Yaskawa INFORM job: u_tourne2TRJ3.JBI

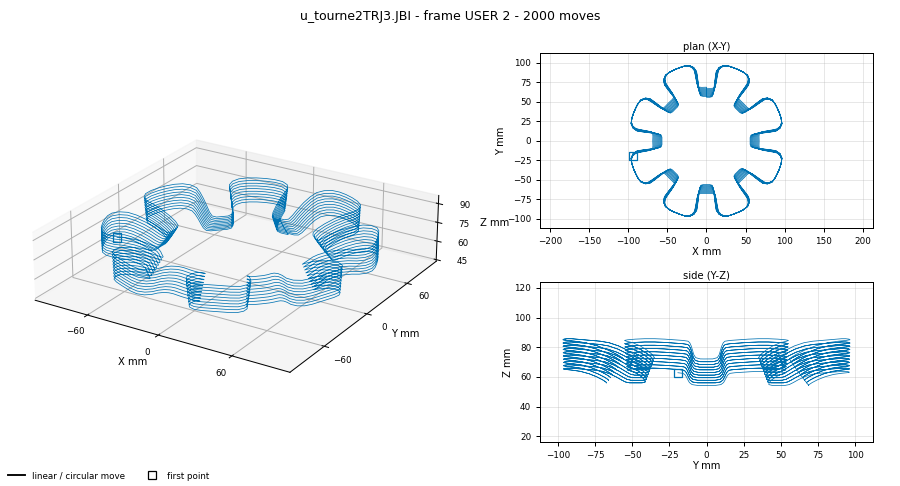
[picture p0: tool path of u_tourne2TRJ3.JBI in frame USER 2, 2000 of 2000 moves have a stored position in this frame; points joined in program order, loops and branches not executed]
/JOB
//NAME u_tourne2TRJ3
///FOLDERNAME DEMO
//POS
///NPOS 2000,0,0,0,0,0
///USER 2
///TOOL 7
///POSTYPE USER
///RECTAN
///RCONF 1,0,0,0,0,0,0,0,0,0,0,0,0,0,0,0,0,0,0,0,0,0,0,0
C00000=-94.423,-19.246,62.877,177.2934,-4.1506,0.0000
C00001=-90.636,-15.942,62.469,172.7027,-3.4329,0.0000
C00002=-85.405,-14.621,61.698,172.2436,-1.7928,0.0000
C00003=-79.780,-13.569,60.151,174.0288,-1.3194,0.0000
C00004=-74.809,-12.586,58.158,176.9959,-0.7631,0.0000
C00005=-71.127,-11.507,56.252,-176.5767,1.2628,0.0000
C00006=-69.044,-9.699,54.888,-163.7827,26.3506,0.0000
C00007=-68.619,-6.200,54.350,-178.9486,38.3072,0.0000
C00008=-68.781,-2.945,54.326,177.7373,38.7538,0.0000
C00009=-68.843,0.000,54.342,180.0000,38.7770,0.0000
C00010=-68.781,2.945,54.326,-177.7373,38.7538,0.0000
C00011=-68.619,6.200,54.350,178.9486,38.3072,0.0000
C00012=-69.044,9.699,54.888,163.7827,26.3559,0.0000
C00013=-71.127,11.507,56.252,176.5767,1.2628,0.0000
C00014=-74.809,12.586,58.158,-176.9959,-0.7631,0.0000
C00015=-79.780,13.569,60.151,-174.0288,-1.3194,0.0000
C00016=-85.405,14.621,61.698,-172.2436,-1.7928,0.0000
C00017=-90.636,15.942,62.469,-172.7027,-3.4329,0.0000
C00018=-94.423,19.246,62.877,-177.2934,-4.1506,0.0000
C00019=-96.154,24.159,63.210,-179.7477,-2.4644,0.0000
C00020=-95.429,29.718,63.547,179.9542,-0.1490,0.0000
C00021=-93.512,35.416,63.770,179.9943,-0.0172,0.0000
C00022=-91.166,41.080,63.770,179.9943,-0.0172,0.0000
C00023=-88.493,46.465,63.547,179.9255,-0.1375,0.0000
C00024=-85.074,50.908,63.210,178.0796,-1.5652,0.0000
C00025=-80.376,53.158,62.877,175.1578,-1.0293,0.0000
C00026=-75.362,52.817,62.469,172.4296,2.7522,0.0000
C00027=-70.729,50.052,61.698,173.2455,4.2443,0.0000
C00028=-66.007,46.818,60.151,174.8393,3.3040,0.0000
C00029=-61.798,43.998,58.158,177.3394,1.5891,0.0000
C00030=-58.431,42.158,56.252,-176.6911,-1.5268,0.0000
C00031=-55.679,41.963,54.888,-150.9263,8.2291,0.0000
C00032=-52.905,44.137,54.350,-150.2465,28.6181,0.0000
C00033=-50.718,46.553,54.326,-151.6440,30.7742,0.0000
C00034=-48.679,48.679,54.342,-150.4041,29.6014,0.0000
C00035=-46.553,50.718,54.326,-149.2258,28.3560,0.0000
C00036=-44.137,52.905,54.350,-151.3819,29.7535,0.0000
C00037=-41.963,55.680,54.888,-171.7709,29.0737,0.0000
C00038=-42.158,58.431,56.252,178.4732,3.3089,0.0000
C00039=-43.998,61.798,58.158,-178.4109,-2.6606,0.0000
C00040=-46.818,66.007,60.151,-176.6960,-5.1607,0.0000
C00041=-50.052,70.729,61.698,-175.7557,-6.7545,0.0000
C00042=-52.817,75.362,62.469,-177.2478,-7.5704,0.0000
C00043=-53.158,80.376,62.877,178.9707,-4.8422,0.0000
C00044=-50.908,85.074,63.210,178.4348,-1.9204,0.0000
C00045=-46.465,88.493,63.547,179.8625,-0.0745,0.0000
C00046=-41.080,91.166,63.770,179.9828,-0.0057,0.0000
C00047=-35.416,93.512,63.770,179.9828,-0.0057,0.0000
C00048=-29.718,95.429,63.547,179.8510,-0.0458,0.0000
C00049=-24.159,96.154,63.210,177.5356,0.2523,0.0000
C00050=-19.246,94.423,62.877,175.8494,2.7066,0.0000
C00051=-15.942,90.636,62.469,176.5671,7.2973,0.0000
C00052=-14.621,85.405,61.698,178.2072,7.7564,0.0000
C00053=-13.569,79.780,60.151,178.6806,5.9712,0.0000
C00054=-12.586,74.809,58.158,179.2369,3.0041,0.0000
C00055=-11.507,71.127,56.252,-178.7372,-3.4233,0.0000
C00056=-9.699,69.044,54.888,-153.6441,-16.2173,0.0000
C00057=-6.200,68.619,54.350,-141.6928,-1.0514,0.0000
C00058=-2.945,68.781,54.326,-141.2462,2.2627,0.0000
C00059=0.000,68.843,54.342,-141.2230,-0.0000,0.0000
C00060=0.000,67.469,56.061,-141.5406,-0.0000,0.0000
C00061=2.820,67.413,56.044,-141.5604,-2.2018,0.0000
C00062=5.989,67.263,56.069,-142.0562,1.4094,0.0000
C00063=9.441,67.734,56.637,-154.9623,16.3637,0.0000
C00064=11.191,69.937,58.076,-179.1454,2.5050,0.0000
C00065=12.227,73.809,60.085,179.1965,-3.3826,0.0000
C00066=13.183,79.025,62.181,178.7265,-6.0864,0.0000
C00067=14.211,84.918,63.804,178.3230,-7.7443,0.0000
C00068=15.500,90.396,64.610,176.7346,-7.3136,0.0000
C00069=18.832,94.373,65.037,175.8895,-2.7812,0.0000
C00070=23.832,96.213,65.385,177.5470,-0.2753,0.0000
C00071=29.513,95.497,65.736,179.8453,0.0458,0.0000
C00072=35.347,93.539,65.969,179.9828,0.0057,0.0000
C00073=41.148,91.136,65.969,179.9828,0.0057,0.0000
C00074=46.658,88.395,65.736,179.8625,0.0745,0.0000
C00075=51.181,84.885,65.385,178.4577,1.9261,0.0000
C00076=53.416,80.048,65.037,179.0569,4.8707,0.0000
C00077=52.959,74.880,64.610,-177.1154,7.4730,0.0000
C00078=49.997,70.095,63.804,-175.6871,6.6682,0.0000
C00079=46.557,65.200,62.181,-176.5862,5.2074,0.0000
C00080=43.545,60.837,60.085,-178.1753,2.9592,0.0000
C00081=41.540,57.367,58.076,178.8300,-2.3790,0.0000
C00082=41.220,54.571,56.637,-173.0071,-28.2766,0.0000
C00083=43.327,51.796,56.069,-151.9011,-29.6258,0.0000
C00084=45.674,49.662,56.044,-149.5306,-28.1040,0.0000
C00085=47.708,47.708,56.061,-150.6808,-29.3192,0.0000
C00086=49.662,45.674,56.044,-151.8960,-30.4694,0.0000
C00087=51.797,43.327,56.069,-150.3742,-28.0989,0.0000
C00088=54.571,41.220,56.637,-151.7234,-6.9929,0.0000
C00089=57.367,41.540,58.076,-177.6210,1.1700,0.0000
C00090=60.837,43.545,60.085,177.0408,-1.8247,0.0000
C00091=65.200,46.557,62.181,174.7926,-3.4138,0.0000
C00092=70.095,49.997,63.804,173.3318,-4.3129,0.0000
C00093=74.880,52.959,64.610,172.5270,-2.8846,0.0000
C00094=80.048,53.416,65.037,175.1293,0.9431,0.0000
C00095=84.885,51.181,65.385,178.0739,1.5423,0.0000
C00096=88.395,46.658,65.736,179.9255,0.1375,0.0000
C00097=91.136,41.148,65.969,179.9943,0.0172,0.0000
C00098=93.539,35.347,65.969,179.9943,0.0172,0.0000
C00099=95.497,29.513,65.736,179.9542,0.1547,0.0000
C00100=96.213,23.832,65.385,-179.7247,2.4530,0.0000
C00101=94.373,18.832,65.037,-177.2188,4.1105,0.0000
C00102=90.396,15.500,64.610,-172.6864,3.2654,0.0000
C00103=84.918,14.211,63.804,-172.2557,1.6770,0.0000
C00104=79.025,13.183,62.181,-173.9136,1.2735,0.0000
C00105=73.809,12.227,60.085,-176.6174,0.8035,0.0000
C00106=69.937,11.191,58.076,177.4950,-0.8546,0.0000
C00107=67.734,9.441,56.637,163.6363,-25.0377,0.0000
C00108=67.263,5.989,56.069,178.5906,-37.9438,0.0000
C00109=67.413,2.820,56.044,-177.7982,-38.4396,0.0000
C00110=67.469,0.000,56.061,-180.0000,-38.4594,0.0000
C00111=67.413,-2.820,56.044,177.7982,-38.4396,0.0000
C00112=67.263,-5.989,56.069,-178.5906,-37.9438,0.0000
C00113=67.734,-9.441,56.637,-163.6363,-25.0377,0.0000
C00114=69.937,-11.191,58.076,-177.4950,-0.8546,0.0000
C00115=73.809,-12.227,60.085,176.6174,0.8035,0.0000
C00116=79.025,-13.183,62.181,173.9136,1.2735,0.0000
C00117=84.918,-14.211,63.804,172.2557,1.6770,0.0000
C00118=90.396,-15.500,64.610,172.6864,3.2654,0.0000
C00119=94.373,-18.832,65.037,177.2188,4.1105,0.0000
C00120=96.213,-23.832,65.385,179.7247,2.4530,0.0000
C00121=95.497,-29.513,65.736,-179.9542,0.1547,0.0000
C00122=93.539,-35.347,65.969,-179.9943,0.0172,0.0000
C00123=91.136,-41.148,65.969,-179.9943,0.0172,0.0000
C00124=88.395,-46.658,65.736,-179.9255,0.1375,0.0000
C00125=84.885,-51.181,65.385,-178.0739,1.5423,0.0000
C00126=80.048,-53.416,65.037,-175.1293,0.9431,0.0000
C00127=74.880,-52.959,64.610,-172.5270,-2.8846,0.0000
C00128=70.095,-49.997,63.804,-173.3318,-4.3129,0.0000
C00129=65.200,-46.557,62.181,-174.7926,-3.4138,0.0000
C00130=60.837,-43.545,60.085,-177.0408,-1.8247,0.0000
C00131=57.367,-41.540,58.076,177.6210,1.1700,0.0000
C00132=54.571,-41.220,56.637,151.7234,-6.9929,0.0000
C00133=51.796,-43.327,56.069,150.3742,-28.0989,0.0000
C00134=49.662,-45.674,56.044,151.8960,-30.4694,0.0000
C00135=47.708,-47.708,56.061,150.6808,-29.3192,0.0000
C00136=45.674,-49.662,56.044,149.5306,-28.1040,0.0000
C00137=43.327,-51.797,56.069,151.9011,-29.6258,0.0000
C00138=41.220,-54.571,56.637,173.0071,-28.2766,0.0000
C00139=41.540,-57.367,58.076,-178.8300,-2.3790,0.0000
C00140=43.545,-60.837,60.085,178.1753,2.9592,0.0000
C00141=46.557,-65.200,62.181,176.5862,5.2074,0.0000
C00142=49.997,-70.095,63.804,175.6871,6.6682,0.0000
C00143=52.959,-74.880,64.610,177.1154,7.4730,0.0000
C00144=53.416,-80.048,65.037,-179.0569,4.8707,0.0000
C00145=51.181,-84.885,65.385,-178.4577,1.9261,0.0000
C00146=46.658,-88.395,65.736,-179.8625,0.0745,0.0000
C00147=41.148,-91.136,65.969,-179.9828,0.0057,0.0000
C00148=35.347,-93.539,65.969,-179.9828,0.0057,0.0000
C00149=29.513,-95.497,65.736,-179.8453,0.0458,0.0000
C00150=23.832,-96.213,65.385,-177.5470,-0.2753,0.0000
C00151=18.832,-94.373,65.037,-175.8895,-2.7812,0.0000
C00152=15.500,-90.396,64.610,-176.7346,-7.3136,0.0000
C00153=14.211,-84.918,63.804,-178.3230,-7.7443,0.0000
C00154=13.183,-79.025,62.181,-178.7265,-6.0864,0.0000
C00155=12.227,-73.809,60.085,-179.1965,-3.3826,0.0000
C00156=11.191,-69.937,58.076,179.1454,2.5050,0.0000
C00157=9.441,-67.734,56.637,154.9623,16.3637,0.0000
C00158=5.989,-67.263,56.069,142.0562,1.4094,0.0000
C00159=2.820,-67.413,56.044,141.5604,-2.2018,0.0000
C00160=0.000,-67.469,56.061,141.5406,-0.0000,0.0000
C00161=0.000,-67.469,56.061,141.5406,-0.0000,0.0000
C00162=-2.820,-67.413,56.044,141.5604,2.2018,0.0000
C00163=-5.989,-67.263,56.069,142.0562,-1.4094,0.0000
C00164=-9.441,-67.734,56.637,154.9623,-16.3637,0.0000
C00165=-11.191,-69.937,58.076,179.1454,-2.5050,0.0000
C00166=-12.227,-73.809,60.085,-179.1965,3.3826,0.0000
C00167=-13.183,-79.025,62.181,-178.7265,6.0864,0.0000
C00168=-14.211,-84.918,63.804,-178.3230,7.7443,0.0000
C00169=-15.500,-90.396,64.610,-176.7346,7.3136,0.0000
C00170=-18.832,-94.373,65.037,-175.8895,2.7812,0.0000
C00171=-23.832,-96.213,65.385,-177.5470,0.2753,0.0000
C00172=-29.513,-95.497,65.736,-179.8453,-0.0458,0.0000
C00173=-35.347,-93.539,65.969,-179.9828,-0.0057,0.0000
C00174=-41.148,-91.136,65.969,-179.9828,-0.0057,0.0000
C00175=-46.658,-88.395,65.736,-179.8625,-0.0745,0.0000
C00176=-51.181,-84.885,65.385,-178.4577,-1.9261,0.0000
C00177=-53.416,-80.048,65.037,-179.0569,-4.8707,0.0000
C00178=-52.959,-74.880,64.610,177.1154,-7.4730,0.0000
C00179=-49.997,-70.095,63.804,175.6871,-6.6682,0.0000
C00180=-46.557,-65.200,62.181,176.5862,-5.2074,0.0000
C00181=-43.545,-60.837,60.085,178.1753,-2.9592,0.0000
C00182=-41.540,-57.367,58.076,-178.8300,2.3790,0.0000
C00183=-41.220,-54.571,56.637,173.0071,28.2766,0.0000
C00184=-43.327,-51.796,56.069,151.9011,29.6258,0.0000
C00185=-45.674,-49.662,56.044,149.5306,28.1040,0.0000
C00186=-47.708,-47.708,56.061,150.6808,29.3192,0.0000
C00187=-49.662,-45.674,56.044,151.8960,30.4694,0.0000
C00188=-51.797,-43.327,56.069,150.3742,28.0989,0.0000
C00189=-54.571,-41.220,56.637,151.7234,6.9929,0.0000
C00190=-57.367,-41.540,58.076,177.6210,-1.1700,0.0000
C00191=-60.837,-43.545,60.085,-177.0408,1.8247,0.0000
C00192=-65.200,-46.557,62.181,-174.7926,3.4138,0.0000
C00193=-70.095,-49.997,63.804,-173.3318,4.3129,0.0000
C00194=-74.880,-52.959,64.610,-172.5270,2.8846,0.0000
C00195=-80.048,-53.416,65.037,-175.1293,-0.9431,0.0000
C00196=-84.885,-51.181,65.385,-178.0739,-1.5423,0.0000
C00197=-88.395,-46.658,65.736,-179.9255,-0.1375,0.0000
C00198=-91.136,-41.148,65.969,-179.9943,-0.0172,0.0000
C00199=-93.539,-35.347,65.969,-179.9943,-0.0172,0.0000
C00200=-95.497,-29.513,65.736,-179.9542,-0.1547,0.0000
C00201=-96.213,-23.832,65.385,179.7247,-2.4530,0.0000
C00202=-94.373,-18.832,65.037,177.2188,-4.1105,0.0000
C00203=-90.396,-15.500,64.610,172.6864,-3.2654,0.0000
C00204=-84.918,-14.211,63.804,172.2557,-1.6770,0.0000
C00205=-79.025,-13.183,62.181,173.9136,-1.2735,0.0000
C00206=-73.809,-12.227,60.085,176.6174,-0.8035,0.0000
C00207=-69.937,-11.191,58.076,-177.4950,0.8546,0.0000
C00208=-67.734,-9.441,56.637,-163.6363,25.0377,0.0000
C00209=-67.263,-5.989,56.069,-178.5906,37.9438,0.0000
C00210=-67.413,-2.820,56.044,177.7982,38.4396,0.0000
C00211=-67.469,0.000,56.061,180.0000,38.4594,0.0000
C00212=-67.413,2.820,56.044,-177.7982,38.4396,0.0000
C00213=-67.263,5.989,56.069,178.5906,37.9438,0.0000
C00214=-67.734,9.441,56.637,163.6363,25.0377,0.0000
C00215=-69.937,11.191,58.076,177.4950,0.8546,0.0000
C00216=-73.809,12.227,60.085,-176.6174,-0.8035,0.0000
C00217=-79.025,13.183,62.181,-173.9136,-1.2735,0.0000
C00218=-84.918,14.211,63.804,-172.2557,-1.6770,0.0000
C00219=-90.396,15.500,64.610,-172.6864,-3.2654,0.0000
C00220=-94.373,18.832,65.037,-177.2188,-4.1105,0.0000
C00221=-96.213,23.832,65.385,-179.7247,-2.4530,0.0000
C00222=-95.497,29.513,65.736,179.9542,-0.1547,0.0000
C00223=-93.539,35.347,65.969,179.9943,-0.0172,0.0000
C00224=-91.136,41.148,65.969,179.9943,-0.0172,0.0000
C00225=-88.395,46.658,65.736,179.9255,-0.1375,0.0000
C00226=-84.885,51.181,65.385,178.0739,-1.5423,0.0000
C00227=-80.048,53.416,65.037,175.1293,-0.9431,0.0000
C00228=-74.880,52.959,64.610,172.5270,2.8846,0.0000
C00229=-70.095,49.997,63.804,173.3318,4.3129,0.0000
C00230=-65.200,46.557,62.181,174.7926,3.4138,0.0000
C00231=-60.837,43.545,60.085,177.0408,1.8247,0.0000
C00232=-57.367,41.540,58.076,-177.6210,-1.1700,0.0000
C00233=-54.571,41.220,56.637,-151.7234,6.9929,0.0000
C00234=-51.796,43.327,56.069,-150.3742,28.0989,0.0000
C00235=-49.662,45.674,56.044,-151.8960,30.4694,0.0000
C00236=-47.708,47.708,56.061,-150.6808,29.3192,0.0000
C00237=-45.674,49.662,56.044,-149.5306,28.1040,0.0000
C00238=-43.327,51.797,56.069,-151.9011,29.6258,0.0000
C00239=-41.220,54.571,56.637,-173.0071,28.2766,0.0000
C00240=-41.540,57.367,58.076,178.8300,2.3790,0.0000
C00241=-43.545,60.837,60.085,-178.1753,-2.9592,0.0000
C00242=-46.557,65.200,62.181,-176.5862,-5.2074,0.0000
C00243=-49.997,70.095,63.804,-175.6871,-6.6682,0.0000
C00244=-52.959,74.880,64.610,-177.1154,-7.4730,0.0000
C00245=-53.416,80.048,65.037,179.0569,-4.8707,0.0000
C00246=-51.181,84.885,65.385,178.4577,-1.9261,0.0000
C00247=-46.658,88.395,65.736,179.8625,-0.0745,0.0000
C00248=-41.148,91.136,65.969,179.9828,-0.0057,0.0000
C00249=-35.347,93.539,65.969,179.9828,-0.0057,0.0000
C00250=-29.513,95.497,65.736,179.8453,-0.0458,0.0000
C00251=-23.832,96.213,65.385,177.5470,0.2753,0.0000
C00252=-18.832,94.373,65.037,175.8895,2.7812,0.0000
C00253=-15.500,90.396,64.610,176.7346,7.3136,0.0000
C00254=-14.211,84.918,63.804,178.3230,7.7443,0.0000
C00255=-13.183,79.025,62.181,178.7265,6.0864,0.0000
C00256=-12.227,73.809,60.085,179.1965,3.3826,0.0000
C00257=-11.191,69.937,58.076,-179.1454,-2.5050,0.0000
C00258=-9.441,67.734,56.637,-154.9623,-16.3637,0.0000
C00259=-5.989,67.263,56.069,-142.0562,-1.4094,0.0000
C00260=-2.820,67.413,56.044,-141.5604,2.2018,0.0000
C00261=0.000,67.469,56.061,-141.5406,-0.0000,0.0000
C00262=0.000,66.107,57.788,-141.9406,-0.0000,0.0000
C00263=2.695,66.055,57.771,-141.9641,-2.1313,0.0000
C00264=5.779,65.917,57.797,-142.5065,1.7619,0.0000
C00265=9.185,66.436,58.394,-156.3339,16.3885,0.0000
C00266=10.880,68.762,59.909,-179.4726,1.6677,0.0000
C00267=11.874,72.826,62.021,179.1732,-3.6871,0.0000
C00268=12.805,78.288,64.219,178.7783,-6.1320,0.0000
C00269=13.814,84.445,65.915,178.4331,-7.6575,0.0000
C00270=15.073,90.163,66.756,176.9144,-7.2602,0.0000
C00271=18.432,94.325,67.200,175.9696,-2.8214,0.0000
C00272=23.517,96.271,67.561,177.5814,-0.2925,0.0000
C00273=29.315,95.562,67.927,179.8510,0.0458,0.0000
C00274=35.280,93.564,68.167,179.9828,0.0057,0.0000
C00275=41.213,91.107,68.167,179.9828,0.0057,0.0000
C00276=46.844,88.301,67.927,179.8625,0.0745,0.0000
C00277=51.445,84.703,67.561,178.4978,1.9147,0.0000
C00278=53.664,79.731,67.200,179.1432,4.8422,0.0000
C00279=53.097,74.413,66.756,-177.0297,7.3058,0.0000
C00280=49.944,69.479,65.915,-175.6707,6.5299,0.0000
C00281=46.303,64.413,64.219,-176.5116,5.2017,0.0000
C00282=43.100,59.892,62.021,-177.9738,3.1951,0.0000
C00283=40.929,56.315,59.909,179.1918,-1.5531,0.0000
C00284=40.483,53.472,58.394,-174.1765,-27.3781,0.0000
C00285=42.524,50.697,57.797,-152.4951,-29.4304,0.0000
C00286=44.802,48.614,57.771,-149.9099,-27.7831,0.0000
C00287=46.745,46.745,57.788,-151.0313,-28.9687,0.0000
C00288=48.613,44.802,57.771,-152.2169,-30.0901,0.0000
C00289=50.697,42.524,57.797,-150.5696,-27.4992,0.0000
C00290=53.472,40.483,58.395,-152.6219,-5.8235,0.0000
C00291=56.315,40.929,59.909,-178.4469,0.8082,0.0000
C00292=59.892,43.100,62.021,176.8049,-2.0262,0.0000
C00293=64.413,46.303,64.219,174.7983,-3.4884,0.0000
C00294=69.479,49.944,65.915,173.4701,-4.3293,0.0000
C00295=74.413,53.097,66.756,172.6942,-2.9703,0.0000
C00296=79.731,53.664,67.200,175.1578,0.8568,0.0000
C00297=84.703,51.445,67.561,178.0853,1.5022,0.0000
C00298=88.301,46.844,67.927,179.9255,0.1375,0.0000
C00299=91.107,41.213,68.167,179.9943,0.0172,0.0000
C00300=93.564,35.280,68.167,179.9943,0.0172,0.0000
C00301=95.562,29.315,67.927,179.9542,0.1490,0.0000
C00302=96.271,23.517,67.561,-179.7075,2.4186,0.0000
C00303=94.325,18.432,67.200,-177.1786,4.0304,0.0000
C00304=90.163,15.073,66.756,-172.7398,3.0856,0.0000
C00305=84.445,13.814,65.915,-172.3425,1.5669,0.0000
C00306=78.288,12.805,64.219,-173.8680,1.2217,0.0000
C00307=72.826,11.874,62.021,-176.3129,0.8268,0.0000
C00308=68.762,10.880,59.909,178.3323,-0.5274,0.0000
C00309=66.436,9.185,58.394,163.6115,-23.6661,0.0000
C00310=65.917,5.779,57.797,178.2381,-37.4935,0.0000
C00311=66.055,2.695,57.771,-177.8687,-38.0359,0.0000
C00312=66.107,0.000,57.788,-180.0000,-38.0594,0.0000
C00313=66.055,-2.695,57.771,177.8687,-38.0359,0.0000
C00314=65.917,-5.780,57.797,-178.2308,-37.4935,0.0000
C00315=66.436,-9.185,58.395,-163.6115,-23.6661,0.0000
C00316=68.762,-10.880,59.909,-178.3323,-0.5274,0.0000
C00317=72.826,-11.874,62.021,176.3129,0.8268,0.0000
C00318=78.288,-12.805,64.219,173.8680,1.2217,0.0000
C00319=84.445,-13.814,65.915,172.3425,1.5669,0.0000
C00320=90.163,-15.073,66.756,172.7398,3.0856,0.0000
C00321=94.325,-18.432,67.200,177.1786,4.0304,0.0000
C00322=96.271,-23.517,67.561,179.7075,2.4186,0.0000
C00323=95.562,-29.315,67.927,-179.9542,0.1490,0.0000
C00324=93.564,-35.280,68.167,-179.9943,0.0172,0.0000
C00325=91.107,-41.213,68.167,-179.9943,0.0172,0.0000
C00326=88.301,-46.844,67.927,-179.9255,0.1375,0.0000
C00327=84.703,-51.445,67.561,-178.0853,1.5022,0.0000
C00328=79.731,-53.664,67.200,-175.1578,0.8568,0.0000
C00329=74.413,-53.097,66.756,-172.6942,-2.9703,0.0000
C00330=69.479,-49.944,65.915,-173.4701,-4.3293,0.0000
C00331=64.413,-46.303,64.219,-174.7983,-3.4884,0.0000
C00332=59.892,-43.100,62.021,-176.8049,-2.0262,0.0000
C00333=56.315,-40.929,59.909,178.4469,0.8082,0.0000
C00334=53.472,-40.483,58.394,152.6219,-5.8235,0.0000
C00335=50.697,-42.524,57.797,150.5696,-27.5049,0.0000
C00336=48.614,-44.802,57.771,152.2169,-30.0901,0.0000
C00337=46.745,-46.745,57.788,151.0313,-28.9687,0.0000
C00338=44.802,-48.613,57.771,149.9099,-27.7831,0.0000
C00339=42.524,-50.697,57.797,152.5008,-29.4304,0.0000
C00340=40.483,-53.472,58.395,174.1765,-27.3781,0.0000
C00341=40.929,-56.315,59.909,-179.1918,-1.5531,0.0000
C00342=43.100,-59.892,62.021,177.9738,3.1951,0.0000
C00343=46.303,-64.413,64.219,176.5116,5.2017,0.0000
C00344=49.944,-69.479,65.915,175.6707,6.5299,0.0000
C00345=53.097,-74.413,66.756,177.0297,7.3058,0.0000
C00346=53.664,-79.731,67.200,-179.1432,4.8422,0.0000
C00347=51.445,-84.703,67.561,-178.4978,1.9147,0.0000
C00348=46.844,-88.301,67.927,-179.8625,0.0745,0.0000
C00349=41.213,-91.107,68.167,-179.9828,0.0057,0.0000
C00350=35.280,-93.564,68.167,-179.9828,0.0057,0.0000
C00351=29.315,-95.562,67.927,-179.8510,0.0458,0.0000
C00352=23.517,-96.271,67.561,-177.5814,-0.2925,0.0000
C00353=18.432,-94.325,67.200,-175.9696,-2.8214,0.0000
C00354=15.073,-90.163,66.756,-176.9144,-7.2602,0.0000
C00355=13.814,-84.445,65.915,-178.4331,-7.6575,0.0000
C00356=12.805,-78.288,64.219,-178.7783,-6.1320,0.0000
C00357=11.874,-72.826,62.021,-179.1732,-3.6871,0.0000
C00358=10.880,-68.762,59.909,179.4726,1.6677,0.0000
C00359=9.185,-66.436,58.394,156.3339,16.3885,0.0000
C00360=5.779,-65.917,57.797,142.5065,1.7619,0.0000
C00361=2.695,-66.055,57.771,141.9641,-2.1313,0.0000
C00362=0.000,-66.107,57.788,141.9406,-0.0000,0.0000
C00363=0.000,-66.107,57.788,141.9406,-0.0000,0.0000
C00364=-2.695,-66.055,57.771,141.9641,2.1313,0.0000
C00365=-5.780,-65.917,57.797,142.5065,-1.7692,0.0000
C00366=-9.185,-66.436,58.395,156.3339,-16.3885,0.0000
C00367=-10.880,-68.762,59.909,179.4726,-1.6677,0.0000
C00368=-11.874,-72.826,62.021,-179.1732,3.6871,0.0000
C00369=-12.805,-78.288,64.219,-178.7783,6.1320,0.0000
C00370=-13.814,-84.445,65.915,-178.4331,7.6575,0.0000
C00371=-15.073,-90.163,66.756,-176.9144,7.2602,0.0000
C00372=-18.432,-94.325,67.200,-175.9696,2.8214,0.0000
C00373=-23.517,-96.271,67.561,-177.5814,0.2925,0.0000
C00374=-29.315,-95.562,67.927,-179.8510,-0.0458,0.0000
C00375=-35.280,-93.564,68.167,-179.9828,-0.0057,0.0000
C00376=-41.213,-91.107,68.167,-179.9828,-0.0057,0.0000
C00377=-46.844,-88.301,67.927,-179.8625,-0.0745,0.0000
C00378=-51.445,-84.703,67.561,-178.4978,-1.9147,0.0000
C00379=-53.664,-79.731,67.200,-179.1432,-4.8422,0.0000
C00380=-53.097,-74.413,66.756,177.0297,-7.3058,0.0000
C00381=-49.944,-69.479,65.915,175.6707,-6.5299,0.0000
C00382=-46.303,-64.413,64.219,176.5116,-5.2017,0.0000
C00383=-43.100,-59.892,62.021,177.9738,-3.1951,0.0000
C00384=-40.929,-56.315,59.909,-179.1918,1.5531,0.0000
C00385=-40.483,-53.472,58.394,174.1765,27.3781,0.0000
C00386=-42.524,-50.697,57.797,152.4951,29.4304,0.0000
C00387=-44.802,-48.614,57.771,149.9099,27.7831,0.0000
C00388=-46.745,-46.745,57.788,151.0313,28.9687,0.0000
C00389=-48.613,-44.802,57.771,152.2169,30.0901,0.0000
C00390=-50.697,-42.524,57.797,150.5696,27.4992,0.0000
C00391=-53.472,-40.483,58.395,152.6219,5.8235,0.0000
C00392=-56.315,-40.929,59.909,178.4469,-0.8082,0.0000
C00393=-59.892,-43.100,62.021,-176.8049,2.0262,0.0000
C00394=-64.413,-46.303,64.219,-174.7983,3.4884,0.0000
C00395=-69.479,-49.944,65.915,-173.4701,4.3293,0.0000
C00396=-74.413,-53.097,66.756,-172.6942,2.9703,0.0000
C00397=-79.731,-53.664,67.200,-175.1578,-0.8568,0.0000
C00398=-84.703,-51.445,67.561,-178.0853,-1.5022,0.0000
C00399=-88.301,-46.844,67.927,-179.9255,-0.1375,0.0000
C00400=-91.107,-41.213,68.167,-179.9943,-0.0172,0.0000
C00401=-93.564,-35.280,68.167,-179.9943,-0.0172,0.0000
C00402=-95.562,-29.315,67.927,-179.9542,-0.1490,0.0000
C00403=-96.271,-23.517,67.561,179.7075,-2.4186,0.0000
C00404=-94.325,-18.432,67.200,177.1786,-4.0304,0.0000
C00405=-90.163,-15.073,66.756,172.7398,-3.0856,0.0000
C00406=-84.445,-13.814,65.915,172.3425,-1.5669,0.0000
C00407=-78.288,-12.805,64.219,173.8680,-1.2217,0.0000
C00408=-72.826,-11.874,62.021,176.3129,-0.8268,0.0000
C00409=-68.762,-10.880,59.909,-178.3323,0.5274,0.0000
C00410=-66.436,-9.185,58.394,-163.6115,23.6661,0.0000
C00411=-65.917,-5.779,57.797,-178.2381,37.4935,0.0000
C00412=-66.055,-2.695,57.771,177.8687,38.0359,0.0000
C00413=-66.107,0.000,57.788,180.0000,38.0594,0.0000
C00414=-66.055,2.695,57.771,-177.8687,38.0359,0.0000
C00415=-65.917,5.780,57.797,178.2308,37.4935,0.0000
C00416=-66.436,9.185,58.395,163.6115,23.6661,0.0000
C00417=-68.762,10.880,59.909,178.3323,0.5274,0.0000
C00418=-72.826,11.874,62.021,-176.3129,-0.8268,0.0000
C00419=-78.288,12.805,64.219,-173.8680,-1.2217,0.0000
C00420=-84.445,13.814,65.915,-172.3425,-1.5669,0.0000
C00421=-90.163,15.073,66.756,-172.7398,-3.0856,0.0000
C00422=-94.325,18.432,67.200,-177.1786,-4.0304,0.0000
C00423=-96.271,23.517,67.561,-179.7075,-2.4186,0.0000
C00424=-95.562,29.315,67.927,179.9542,-0.1490,0.0000
C00425=-93.564,35.280,68.167,179.9943,-0.0172,0.0000
C00426=-91.107,41.213,68.167,179.9943,-0.0172,0.0000
C00427=-88.301,46.844,67.927,179.9255,-0.1375,0.0000
C00428=-84.703,51.445,67.561,178.0853,-1.5022,0.0000
C00429=-79.731,53.664,67.200,175.1578,-0.8568,0.0000
C00430=-74.413,53.097,66.756,172.6942,2.9703,0.0000
C00431=-69.479,49.944,65.915,173.4701,4.3293,0.0000
C00432=-64.413,46.303,64.219,174.7983,3.4884,0.0000
C00433=-59.892,43.100,62.021,176.8049,2.0262,0.0000
C00434=-56.315,40.929,59.909,-178.4469,-0.8082,0.0000
C00435=-53.472,40.483,58.394,-152.6219,5.8235,0.0000
C00436=-50.697,42.524,57.797,-150.5696,27.5049,0.0000
C00437=-48.614,44.802,57.771,-152.2169,30.0901,0.0000
C00438=-46.745,46.745,57.788,-151.0313,28.9687,0.0000
C00439=-44.802,48.613,57.771,-149.9099,27.7831,0.0000
C00440=-42.524,50.697,57.797,-152.5008,29.4304,0.0000
C00441=-40.483,53.472,58.395,-174.1765,27.3781,0.0000
C00442=-40.929,56.315,59.909,179.1918,1.5531,0.0000
C00443=-43.100,59.892,62.021,-177.9738,-3.1951,0.0000
C00444=-46.303,64.413,64.219,-176.5116,-5.2017,0.0000
C00445=-49.944,69.479,65.915,-175.6707,-6.5299,0.0000
C00446=-53.097,74.413,66.756,-177.0297,-7.3058,0.0000
C00447=-53.664,79.731,67.200,179.1432,-4.8422,0.0000
C00448=-51.445,84.703,67.561,178.4978,-1.9147,0.0000
C00449=-46.844,88.301,67.927,179.8625,-0.0745,0.0000
C00450=-41.213,91.107,68.167,179.9828,-0.0057,0.0000
C00451=-35.280,93.564,68.167,179.9828,-0.0057,0.0000
C00452=-29.315,95.562,67.927,179.8510,-0.0458,0.0000
C00453=-23.517,96.271,67.561,177.5814,0.2925,0.0000
C00454=-18.432,94.325,67.200,175.9696,2.8214,0.0000
C00455=-15.073,90.163,66.756,176.9144,7.2602,0.0000
C00456=-13.814,84.445,65.915,178.4331,7.6575,0.0000
C00457=-12.805,78.288,64.219,178.7783,6.1320,0.0000
C00458=-11.874,72.826,62.021,179.1732,3.6871,0.0000
C00459=-10.880,68.762,59.909,-179.4726,-1.6677,0.0000
C00460=-9.185,66.436,58.395,-156.3339,-16.3885,0.0000
C00461=-5.780,65.917,57.797,-142.5065,-1.7692,0.0000
C00462=-2.695,66.055,57.771,-141.9641,2.1313,0.0000
C00463=0.000,66.107,57.788,-141.9406,-0.0000,0.0000
C00464=0.000,64.758,59.526,-142.4265,-0.0000,0.0000
C00465=2.572,64.710,59.508,-142.4457,-2.0524,0.0000
C00466=5.572,64.584,59.535,-143.0521,2.1078,0.0000
C00467=8.932,65.152,60.163,-157.7445,16.2794,0.0000
C00468=10.572,67.603,61.754,-179.7307,0.9110,0.0000
C00469=11.527,71.864,63.969,179.1672,-3.9284,0.0000
C00470=12.439,77.571,66.266,178.8417,-6.1206,0.0000
C00471=13.430,83.988,68.033,178.5493,-7.5068,0.0000
C00472=14.662,89.940,68.906,177.1001,-7.1264,0.0000
C00473=18.048,94.279,69.366,176.0905,-2.8266,0.0000
C00474=23.215,96.325,69.740,177.6386,-0.3039,0.0000
C00475=29.126,95.625,70.117,179.8510,0.0458,0.0000
C00476=35.216,93.589,70.366,179.9828,0.0057,0.0000
C00477=41.276,91.079,70.366,179.9828,0.0057,0.0000
C00478=47.022,88.212,70.117,179.8625,0.0745,0.0000
C00479=51.697,84.528,69.740,178.5437,1.8803,0.0000
C00480=53.903,79.427,69.366,179.2296,4.7613,0.0000
C00481=53.229,73.964,68.906,-176.9848,7.0809,0.0000
C00482=49.892,68.885,68.033,-175.6955,6.3389,0.0000
C00483=46.056,63.647,66.266,-176.4771,5.1503,0.0000
C00484=42.664,58.966,63.969,-177.8126,3.3678,0.0000
C00485=40.327,55.279,61.754,179.5416,-0.8365,0.0000
C00486=39.754,52.385,60.163,-175.2650,-26.3749,0.0000
C00487=41.728,49.608,59.535,-153.1659,-29.1544,0.0000
C00488=43.938,47.576,59.508,-150.3619,-27.3947,0.0000
C00489=45.791,45.791,59.526,-151.4524,-28.5476,0.0000
C00490=47.575,43.938,59.508,-152.6053,-29.6381,0.0000
C00491=49.608,41.728,59.535,-150.8401,-26.8284,0.0000
C00492=52.385,39.754,60.163,-153.6251,-4.7350,0.0000
C00493=55.279,40.327,61.754,-179.1635,0.4584,0.0000
C00494=58.966,42.664,63.969,176.6322,-2.1874,0.0000
C00495=63.647,46.056,66.266,174.8497,-3.5229,0.0000
C00496=68.885,49.892,68.033,173.6611,-4.3045,0.0000
C00497=73.964,53.229,68.906,172.9191,-3.0152,0.0000
C00498=79.427,53.903,69.366,175.2387,0.7704,0.0000
C00499=84.528,51.697,69.740,178.1197,1.4563,0.0000
C00500=88.212,47.022,70.117,179.9255,0.1375,0.0000
C00501=91.079,41.276,70.366,179.9943,0.0172,0.0000
C00502=93.589,35.216,70.366,179.9943,0.0172,0.0000
C00503=95.625,29.126,70.117,179.9542,0.1490,0.0000
C00504=96.325,23.215,69.740,-179.6961,2.3614,0.0000
C00505=94.279,18.048,69.366,-177.1734,3.9095,0.0000
C00506=89.940,14.662,68.906,-172.8736,2.8999,0.0000
C00507=83.988,13.430,68.033,-172.4932,1.4507,0.0000
C00508=77.571,12.439,66.266,-173.8794,1.1583,0.0000
C00509=71.864,11.527,63.969,-176.0716,0.8328,0.0000
C00510=67.603,10.572,61.754,179.0890,-0.2693,0.0000
C00511=65.152,8.932,60.163,163.7206,-22.2555,0.0000
C00512=64.584,5.572,59.535,177.8922,-36.9479,0.0000
C00513=64.710,2.572,59.508,-177.9476,-37.5543,0.0000
C00514=64.758,0.000,59.526,-180.0000,-37.5735,0.0000
C00515=64.710,-2.572,59.508,177.9476,-37.5543,0.0000
C00516=64.584,-5.572,59.535,-177.8922,-36.9479,0.0000
C00517=65.152,-8.932,60.163,-163.7206,-22.2555,0.0000
C00518=67.603,-10.572,61.754,-179.0890,-0.2693,0.0000
C00519=71.864,-11.527,63.969,176.0716,0.8328,0.0000
C00520=77.571,-12.439,66.266,173.8794,1.1583,0.0000
C00521=83.988,-13.430,68.033,172.4932,1.4507,0.0000
C00522=89.940,-14.662,68.906,172.8736,2.8999,0.0000
C00523=94.279,-18.048,69.366,177.1734,3.9095,0.0000
C00524=96.325,-23.215,69.740,179.6961,2.3614,0.0000
C00525=95.625,-29.126,70.117,-179.9542,0.1490,0.0000
C00526=93.589,-35.216,70.366,-179.9943,0.0172,0.0000
C00527=91.079,-41.276,70.366,-179.9943,0.0172,0.0000
C00528=88.212,-47.022,70.117,-179.9255,0.1375,0.0000
C00529=84.528,-51.697,69.740,-178.1197,1.4563,0.0000
C00530=79.427,-53.903,69.366,-175.2387,0.7704,0.0000
C00531=73.964,-53.229,68.906,-172.9191,-3.0152,0.0000
C00532=68.885,-49.892,68.033,-173.6611,-4.3045,0.0000
C00533=63.647,-46.056,66.266,-174.8497,-3.5229,0.0000
C00534=58.966,-42.664,63.969,-176.6322,-2.1874,0.0000
C00535=55.279,-40.327,61.754,179.1635,0.4584,0.0000
C00536=52.385,-39.754,60.163,153.6251,-4.7350,0.0000
C00537=49.608,-41.728,59.535,150.8456,-26.8341,0.0000
C00538=47.576,-43.938,59.508,152.6053,-29.6381,0.0000
C00539=45.791,-45.791,59.526,151.4524,-28.5476,0.0000
C00540=43.938,-47.575,59.508,150.3619,-27.3947,0.0000
C00541=41.728,-49.608,59.535,153.1716,-29.1599,0.0000
C00542=39.754,-52.385,60.163,175.2650,-26.3749,0.0000
C00543=40.327,-55.279,61.754,-179.5416,-0.8365,0.0000
C00544=42.664,-58.966,63.969,177.8126,3.3678,0.0000
C00545=46.056,-63.647,66.266,176.4771,5.1503,0.0000
C00546=49.892,-68.885,68.033,175.6955,6.3389,0.0000
C00547=53.229,-73.964,68.906,176.9848,7.0809,0.0000
C00548=53.903,-79.427,69.366,-179.2296,4.7613,0.0000
C00549=51.697,-84.528,69.740,-178.5437,1.8803,0.0000
C00550=47.022,-88.212,70.117,-179.8625,0.0745,0.0000
C00551=41.276,-91.079,70.366,-179.9828,0.0057,0.0000
C00552=35.216,-93.589,70.366,-179.9828,0.0057,0.0000
C00553=29.126,-95.625,70.117,-179.8510,0.0458,0.0000
C00554=23.215,-96.325,69.740,-177.6386,-0.3039,0.0000
C00555=18.048,-94.279,69.366,-176.0905,-2.8266,0.0000
C00556=14.662,-89.940,68.906,-177.1001,-7.1264,0.0000
C00557=13.430,-83.988,68.033,-178.5493,-7.5068,0.0000
C00558=12.439,-77.571,66.266,-178.8417,-6.1206,0.0000
C00559=11.527,-71.864,63.969,-179.1672,-3.9284,0.0000
C00560=10.572,-67.603,61.754,179.7307,0.9110,0.0000
C00561=8.932,-65.152,60.163,157.7445,16.2794,0.0000
C00562=5.572,-64.584,59.535,143.0521,2.1078,0.0000
C00563=2.572,-64.710,59.508,142.4457,-2.0524,0.0000
C00564=0.000,-64.758,59.526,142.4265,-0.0000,0.0000
C00565=0.000,-64.758,59.526,142.4265,-0.0000,0.0000
C00566=-2.572,-64.710,59.508,142.4457,2.0524,0.0000
C00567=-5.572,-64.584,59.535,143.0521,-2.1078,0.0000
C00568=-8.932,-65.152,60.163,157.7445,-16.2794,0.0000
C00569=-10.572,-67.603,61.754,179.7307,-0.9110,0.0000
C00570=-11.527,-71.864,63.969,-179.1672,3.9284,0.0000
C00571=-12.439,-77.571,66.266,-178.8417,6.1206,0.0000
C00572=-13.430,-83.988,68.033,-178.5493,7.5068,0.0000
C00573=-14.662,-89.940,68.906,-177.1001,7.1264,0.0000
C00574=-18.048,-94.279,69.366,-176.0905,2.8266,0.0000
C00575=-23.215,-96.325,69.740,-177.6386,0.3039,0.0000
C00576=-29.126,-95.625,70.117,-179.8510,-0.0458,0.0000
C00577=-35.216,-93.589,70.366,-179.9828,-0.0057,0.0000
C00578=-41.276,-91.079,70.366,-179.9828,-0.0057,0.0000
C00579=-47.022,-88.212,70.117,-179.8625,-0.0745,0.0000
C00580=-51.697,-84.528,69.740,-178.5437,-1.8803,0.0000
C00581=-53.903,-79.427,69.366,-179.2296,-4.7613,0.0000
C00582=-53.229,-73.964,68.906,176.9848,-7.0809,0.0000
C00583=-49.892,-68.885,68.033,175.6955,-6.3389,0.0000
C00584=-46.056,-63.647,66.266,176.4771,-5.1503,0.0000
C00585=-42.664,-58.966,63.969,177.8126,-3.3678,0.0000
C00586=-40.327,-55.279,61.754,-179.5416,0.8365,0.0000
C00587=-39.754,-52.385,60.163,175.2650,26.3749,0.0000
C00588=-41.728,-49.608,59.535,153.1659,29.1544,0.0000
C00589=-43.938,-47.576,59.508,150.3619,27.3947,0.0000
C00590=-45.791,-45.791,59.526,151.4524,28.5476,0.0000
C00591=-47.575,-43.938,59.508,152.6053,29.6381,0.0000
C00592=-49.608,-41.728,59.535,150.8401,26.8284,0.0000
C00593=-52.385,-39.754,60.163,153.6251,4.7350,0.0000
C00594=-55.279,-40.327,61.754,179.1635,-0.4584,0.0000
C00595=-58.966,-42.664,63.969,-176.6322,2.1874,0.0000
C00596=-63.647,-46.056,66.266,-174.8497,3.5229,0.0000
C00597=-68.885,-49.892,68.033,-173.6611,4.3045,0.0000
C00598=-73.964,-53.229,68.906,-172.9191,3.0152,0.0000
C00599=-79.427,-53.903,69.366,-175.2387,-0.7704,0.0000
C00600=-84.528,-51.697,69.740,-178.1197,-1.4563,0.0000
C00601=-88.212,-47.022,70.117,-179.9255,-0.1375,0.0000
C00602=-91.079,-41.276,70.366,-179.9943,-0.0172,0.0000
C00603=-93.589,-35.216,70.366,-179.9943,-0.0172,0.0000
C00604=-95.625,-29.126,70.117,-179.9542,-0.1490,0.0000
C00605=-96.325,-23.215,69.740,179.6961,-2.3614,0.0000
C00606=-94.279,-18.048,69.366,177.1734,-3.9095,0.0000
C00607=-89.940,-14.662,68.906,172.8736,-2.8999,0.0000
C00608=-83.988,-13.430,68.033,172.4932,-1.4507,0.0000
C00609=-77.571,-12.439,66.266,173.8794,-1.1583,0.0000
C00610=-71.864,-11.527,63.969,176.0716,-0.8328,0.0000
C00611=-67.603,-10.572,61.754,-179.0890,0.2693,0.0000
C00612=-65.152,-8.932,60.163,-163.7206,22.2555,0.0000
C00613=-64.584,-5.572,59.535,-177.8922,36.9479,0.0000
C00614=-64.710,-2.572,59.508,177.9476,37.5543,0.0000
C00615=-64.758,0.000,59.526,180.0000,37.5735,0.0000
C00616=-64.710,2.572,59.508,-177.9476,37.5543,0.0000
C00617=-64.584,5.572,59.535,177.8922,36.9479,0.0000
C00618=-65.152,8.932,60.163,163.7206,22.2555,0.0000
C00619=-67.603,10.572,61.754,179.0890,0.2693,0.0000
C00620=-71.864,11.527,63.969,-176.0716,-0.8328,0.0000
C00621=-77.571,12.439,66.266,-173.8794,-1.1583,0.0000
C00622=-83.988,13.430,68.033,-172.4932,-1.4507,0.0000
C00623=-89.940,14.662,68.906,-172.8736,-2.8999,0.0000
C00624=-94.279,18.048,69.366,-177.1734,-3.9095,0.0000
C00625=-96.325,23.215,69.740,-179.6961,-2.3614,0.0000
C00626=-95.625,29.126,70.117,179.9542,-0.1490,0.0000
C00627=-93.589,35.216,70.366,179.9943,-0.0172,0.0000
C00628=-91.079,41.276,70.366,179.9943,-0.0172,0.0000
C00629=-88.212,47.022,70.117,179.9255,-0.1375,0.0000
C00630=-84.528,51.697,69.740,178.1197,-1.4563,0.0000
C00631=-79.427,53.903,69.366,175.2387,-0.7704,0.0000
C00632=-73.964,53.229,68.906,172.9191,3.0152,0.0000
C00633=-68.885,49.892,68.033,173.6611,4.3045,0.0000
C00634=-63.647,46.056,66.266,174.8497,3.5229,0.0000
C00635=-58.966,42.664,63.969,176.6322,2.1874,0.0000
C00636=-55.279,40.327,61.754,-179.1635,-0.4584,0.0000
C00637=-52.385,39.754,60.163,-153.6251,4.7350,0.0000
C00638=-49.608,41.728,59.535,-150.8456,26.8341,0.0000
C00639=-47.576,43.938,59.508,-152.6053,29.6381,0.0000
C00640=-45.791,45.791,59.526,-151.4524,28.5476,0.0000
C00641=-43.938,47.575,59.508,-150.3619,27.3947,0.0000
C00642=-41.728,49.608,59.535,-153.1716,29.1599,0.0000
C00643=-39.754,52.385,60.163,-175.2650,26.3749,0.0000
C00644=-40.327,55.279,61.754,179.5416,0.8365,0.0000
C00645=-42.664,58.966,63.969,-177.8126,-3.3678,0.0000
C00646=-46.056,63.647,66.266,-176.4771,-5.1503,0.0000
C00647=-49.892,68.885,68.033,-175.6955,-6.3389,0.0000
C00648=-53.229,73.964,68.906,-176.9848,-7.0809,0.0000
C00649=-53.903,79.427,69.366,179.2296,-4.7613,0.0000
C00650=-51.697,84.528,69.740,178.5437,-1.8803,0.0000
C00651=-47.022,88.212,70.117,179.8625,-0.0745,0.0000
C00652=-41.276,91.079,70.366,179.9828,-0.0057,0.0000
C00653=-35.216,93.589,70.366,179.9828,-0.0057,0.0000
C00654=-29.126,95.625,70.117,179.8510,-0.0458,0.0000
C00655=-23.215,96.325,69.740,177.6386,0.3039,0.0000
C00656=-18.048,94.279,69.366,176.0905,2.8266,0.0000
C00657=-14.662,89.940,68.906,177.1001,7.1264,0.0000
C00658=-13.430,83.988,68.033,178.5493,7.5068,0.0000
C00659=-12.439,77.571,66.266,178.8417,6.1206,0.0000
C00660=-11.527,71.864,63.969,179.1672,3.9284,0.0000
C00661=-10.572,67.603,61.754,-179.7307,-0.9110,0.0000
C00662=-8.932,65.152,60.163,-157.7445,-16.2794,0.0000
C00663=-5.572,64.584,59.535,-143.0521,-2.1078,0.0000
C00664=-2.572,64.710,59.508,-142.4457,2.0524,0.0000
C00665=0.000,64.758,59.526,-142.4265,-0.0000,0.0000
C00666=0.000,63.425,61.276,-142.9995,-0.0000,0.0000
C00667=2.450,63.381,61.257,-143.0189,-1.9725,0.0000
C00668=5.367,63.268,61.285,-143.6885,2.4389,0.0000
C00669=8.682,63.886,61.945,-159.1759,16.0518,0.0000
C00670=10.270,66.465,63.612,-179.9370,0.2406,0.0000
C00671=11.189,70.924,65.929,179.1728,-4.1007,0.0000
C00672=12.084,76.878,68.324,178.9053,-6.0453,0.0000
C00673=13.063,83.550,70.157,178.6599,-7.2864,0.0000
C00674=14.270,89.726,71.060,177.2978,-6.9230,0.0000
C00675=17.683,94.235,71.535,176.2458,-2.7916,0.0000
C00676=22.929,96.378,71.920,177.7247,-0.3096,0.0000
C00677=28.946,95.684,72.309,179.8568,0.0401,0.0000
C00678=35.156,93.612,72.565,179.9828,0.0057,0.0000
C00679=41.335,91.053,72.565,179.9828,0.0057,0.0000
C00680=47.191,88.127,72.309,179.8682,0.0745,0.0000
C00681=51.936,84.362,71.920,178.6069,1.8286,0.0000
C00682=54.130,79.138,71.535,179.3160,4.6290,0.0000
C00683=53.356,73.536,71.060,-176.9924,6.7977,0.0000
C00684=49.842,68.316,70.157,-175.7728,6.1010,0.0000
C00685=45.816,62.906,68.324,-176.4893,5.0463,0.0000
C00686=42.239,58.063,65.929,-177.6803,3.4830,0.0000
C00687=39.736,54.260,63.612,179.8739,-0.2177,0.0000
C00688=39.035,51.313,61.945,-176.2538,-25.2815,0.0000
C00689=40.942,48.532,61.285,-153.9179,-28.7990,0.0000
C00690=43.085,46.550,61.257,-150.8912,-26.9398,0.0000
C00691=44.848,44.848,61.276,-151.9510,-28.0490,0.0000
C00692=46.550,43.085,61.257,-153.0602,-29.1088,0.0000
C00693=48.532,40.942,61.285,-151.2010,-26.0821,0.0000
C00694=51.313,39.035,61.945,-154.7185,-3.7462,0.0000
C00695=54.260,39.736,63.612,-179.7823,0.1261,0.0000
C00696=58.063,42.239,65.929,176.5170,-2.3197,0.0000
C00697=62.906,45.816,68.324,174.9537,-3.5107,0.0000
C00698=68.316,49.842,70.157,173.8990,-4.2272,0.0000
C00699=73.536,53.356,71.060,173.2023,-3.0076,0.0000
C00700=79.138,54.130,71.535,175.3710,0.6840,0.0000
C00701=84.362,51.936,71.920,178.1714,1.3931,0.0000
C00702=88.127,47.191,72.309,179.9255,0.1318,0.0000
C00703=91.053,41.335,72.565,179.9943,0.0172,0.0000
C00704=93.612,35.156,72.565,179.9943,0.0172,0.0000
C00705=95.684,28.946,72.309,179.9599,0.1432,0.0000
C00706=96.378,22.929,71.920,-179.6904,2.2753,0.0000
C00707=94.235,17.683,71.535,-177.2084,3.7542,0.0000
C00708=89.726,14.270,71.060,-173.0770,2.7022,0.0000
C00709=83.550,13.063,70.157,-172.7136,1.3401,0.0000
C00710=76.878,12.084,68.324,-173.9547,1.0947,0.0000
C00711=70.924,11.189,65.929,-175.8993,0.8272,0.0000
C00712=66.465,10.270,63.612,179.7594,-0.0630,0.0000
C00713=63.886,8.682,61.945,163.9482,-20.8241,0.0000
C00714=63.268,5.367,61.285,177.5611,-36.3115,0.0000
C00715=63.381,2.450,61.257,-178.0275,-36.9811,0.0000
C00716=63.425,0.000,61.276,-180.0000,-37.0005,0.0000
C00717=63.381,-2.450,61.257,178.0275,-36.9811,0.0000
C00718=63.268,-5.367,61.285,-177.5611,-36.3115,0.0000
C00719=63.886,-8.682,61.945,-163.9482,-20.8185,0.0000
C00720=66.465,-10.270,63.612,-179.7594,-0.0630,0.0000
C00721=70.924,-11.189,65.929,175.8993,0.8272,0.0000
C00722=76.878,-12.084,68.324,173.9547,1.0947,0.0000
C00723=83.550,-13.063,70.157,172.7136,1.3401,0.0000
C00724=89.726,-14.270,71.060,173.0770,2.7022,0.0000
C00725=94.235,-17.683,71.535,177.2084,3.7542,0.0000
C00726=96.378,-22.929,71.920,179.6904,2.2753,0.0000
C00727=95.684,-28.946,72.309,-179.9599,0.1432,0.0000
C00728=93.612,-35.156,72.565,-179.9943,0.0172,0.0000
C00729=91.053,-41.335,72.565,-179.9943,0.0172,0.0000
C00730=88.127,-47.191,72.309,-179.9255,0.1318,0.0000
C00731=84.362,-51.936,71.920,-178.1714,1.3931,0.0000
C00732=79.138,-54.130,71.535,-175.3710,0.6840,0.0000
C00733=73.536,-53.356,71.060,-173.2023,-3.0076,0.0000
C00734=68.316,-49.842,70.157,-173.8990,-4.2272,0.0000
C00735=62.906,-45.816,68.324,-174.9537,-3.5107,0.0000
C00736=58.063,-42.239,65.929,-176.5170,-2.3197,0.0000
C00737=54.260,-39.736,63.612,179.7823,0.1261,0.0000
C00738=51.313,-39.035,61.945,154.7185,-3.7462,0.0000
C00739=48.532,-40.942,61.285,151.2010,-26.0821,0.0000
C00740=46.550,-43.085,61.257,153.0602,-29.1088,0.0000
C00741=44.848,-44.848,61.276,151.9510,-28.0490,0.0000
C00742=43.085,-46.550,61.257,150.8912,-26.9398,0.0000
C00743=40.942,-48.532,61.285,153.9179,-28.7990,0.0000
C00744=39.035,-51.313,61.945,176.2538,-25.2815,0.0000
C00745=39.736,-54.260,63.612,-179.8739,-0.2177,0.0000
C00746=42.239,-58.063,65.929,177.6803,3.4830,0.0000
C00747=45.816,-62.906,68.324,176.4893,5.0463,0.0000
C00748=49.842,-68.316,70.157,175.7728,6.1010,0.0000
C00749=53.356,-73.536,71.060,176.9924,6.7977,0.0000
C00750=54.130,-79.138,71.535,-179.3160,4.6290,0.0000
C00751=51.936,-84.362,71.920,-178.6069,1.8286,0.0000
C00752=47.191,-88.127,72.309,-179.8682,0.0745,0.0000
C00753=41.335,-91.053,72.565,-179.9828,0.0057,0.0000
C00754=35.156,-93.612,72.565,-179.9828,0.0057,0.0000
C00755=28.946,-95.684,72.309,-179.8568,0.0401,0.0000
C00756=22.929,-96.378,71.920,-177.7247,-0.3096,0.0000
C00757=17.683,-94.235,71.535,-176.2458,-2.7916,0.0000
C00758=14.270,-89.726,71.060,-177.2978,-6.9230,0.0000
C00759=13.063,-83.550,70.157,-178.6599,-7.2864,0.0000
C00760=12.084,-76.878,68.324,-178.9053,-6.0453,0.0000
C00761=11.189,-70.924,65.929,-179.1728,-4.1007,0.0000
C00762=10.270,-66.465,63.612,179.9370,0.2406,0.0000
C00763=8.682,-63.886,61.945,159.1759,16.0518,0.0000
C00764=5.367,-63.268,61.285,143.6885,2.4389,0.0000
C00765=2.450,-63.381,61.257,143.0189,-1.9725,0.0000
C00766=0.000,-63.425,61.276,142.9995,-0.0000,0.0000
C00767=0.000,-63.425,61.276,142.9995,-0.0000,0.0000
C00768=-2.450,-63.381,61.257,143.0189,1.9725,0.0000
C00769=-5.367,-63.268,61.285,143.6885,-2.4389,0.0000
C00770=-8.682,-63.886,61.945,159.1815,-16.0518,0.0000
C00771=-10.270,-66.465,63.612,179.9370,-0.2406,0.0000
C00772=-11.189,-70.924,65.929,-179.1728,4.1007,0.0000
C00773=-12.084,-76.878,68.324,-178.9053,6.0453,0.0000
C00774=-13.063,-83.550,70.157,-178.6599,7.2864,0.0000
C00775=-14.270,-89.726,71.060,-177.2978,6.9230,0.0000
C00776=-17.683,-94.235,71.535,-176.2458,2.7916,0.0000
C00777=-22.929,-96.378,71.920,-177.7247,0.3096,0.0000
C00778=-28.946,-95.684,72.309,-179.8568,-0.0401,0.0000
C00779=-35.156,-93.612,72.565,-179.9828,-0.0057,0.0000
C00780=-41.335,-91.053,72.565,-179.9828,-0.0057,0.0000
C00781=-47.191,-88.127,72.309,-179.8682,-0.0745,0.0000
C00782=-51.936,-84.362,71.920,-178.6069,-1.8286,0.0000
C00783=-54.130,-79.138,71.535,-179.3160,-4.6290,0.0000
C00784=-53.356,-73.536,71.060,176.9924,-6.7977,0.0000
C00785=-49.842,-68.316,70.157,175.7728,-6.1010,0.0000
C00786=-45.816,-62.906,68.324,176.4893,-5.0463,0.0000
C00787=-42.239,-58.063,65.929,177.6803,-3.4830,0.0000
C00788=-39.736,-54.260,63.612,-179.8739,0.2177,0.0000
C00789=-39.035,-51.313,61.945,176.2538,25.2815,0.0000
C00790=-40.942,-48.532,61.285,153.9179,28.7990,0.0000
C00791=-43.085,-46.550,61.257,150.8912,26.9398,0.0000
C00792=-44.848,-44.848,61.276,151.9510,28.0490,0.0000
C00793=-46.550,-43.085,61.257,153.0602,29.1088,0.0000
C00794=-48.532,-40.942,61.285,151.2010,26.0821,0.0000
C00795=-51.313,-39.035,61.945,154.7185,3.7462,0.0000
C00796=-54.260,-39.736,63.612,179.7823,-0.1261,0.0000
C00797=-58.063,-42.239,65.929,-176.5170,2.3197,0.0000
C00798=-62.906,-45.816,68.324,-174.9537,3.5107,0.0000
C00799=-68.316,-49.842,70.157,-173.8990,4.2272,0.0000
C00800=-73.536,-53.356,71.060,-173.2023,3.0076,0.0000
C00801=-79.138,-54.130,71.535,-175.3710,-0.6840,0.0000
C00802=-84.362,-51.936,71.920,-178.1714,-1.3931,0.0000
C00803=-88.127,-47.191,72.309,-179.9255,-0.1318,0.0000
C00804=-91.053,-41.335,72.565,-179.9943,-0.0172,0.0000
C00805=-93.612,-35.156,72.565,-179.9943,-0.0172,0.0000
C00806=-95.684,-28.946,72.309,-179.9599,-0.1432,0.0000
C00807=-96.378,-22.929,71.920,179.6904,-2.2753,0.0000
C00808=-94.235,-17.683,71.535,177.2084,-3.7542,0.0000
C00809=-89.726,-14.270,71.060,173.0770,-2.7022,0.0000
C00810=-83.550,-13.063,70.157,172.7136,-1.3401,0.0000
C00811=-76.878,-12.084,68.324,173.9547,-1.0947,0.0000
C00812=-70.924,-11.189,65.929,175.8993,-0.8272,0.0000
C00813=-66.465,-10.270,63.612,-179.7594,0.0630,0.0000
C00814=-63.886,-8.682,61.945,-163.9482,20.8241,0.0000
C00815=-63.268,-5.367,61.285,-177.5611,36.3115,0.0000
C00816=-63.381,-2.450,61.257,178.0275,36.9811,0.0000
C00817=-63.425,0.000,61.276,180.0000,37.0005,0.0000
C00818=-63.381,2.450,61.257,-178.0275,36.9811,0.0000
C00819=-63.268,5.367,61.285,177.5611,36.3115,0.0000
C00820=-63.886,8.682,61.945,163.9482,20.8185,0.0000
C00821=-66.465,10.270,63.612,179.7594,0.0630,0.0000
C00822=-70.924,11.189,65.929,-175.8993,-0.8272,0.0000
C00823=-76.878,12.084,68.324,-173.9547,-1.0947,0.0000
C00824=-83.550,13.063,70.157,-172.7136,-1.3401,0.0000
C00825=-89.726,14.270,71.060,-173.0770,-2.7022,0.0000
C00826=-94.235,17.683,71.535,-177.2084,-3.7542,0.0000
C00827=-96.378,22.929,71.920,-179.6904,-2.2753,0.0000
C00828=-95.684,28.946,72.309,179.9599,-0.1432,0.0000
C00829=-93.612,35.156,72.565,179.9943,-0.0172,0.0000
C00830=-91.053,41.335,72.565,179.9943,-0.0172,0.0000
C00831=-88.127,47.191,72.309,179.9255,-0.1318,0.0000
C00832=-84.362,51.936,71.920,178.1714,-1.3931,0.0000
C00833=-79.138,54.130,71.535,175.3710,-0.6840,0.0000
C00834=-73.536,53.356,71.060,173.2023,3.0076,0.0000
C00835=-68.316,49.842,70.157,173.8990,4.2272,0.0000
C00836=-62.906,45.816,68.324,174.9537,3.5107,0.0000
C00837=-58.063,42.239,65.929,176.5170,2.3197,0.0000
C00838=-54.260,39.736,63.612,-179.7823,-0.1261,0.0000
C00839=-51.313,39.035,61.945,-154.7185,3.7462,0.0000
C00840=-48.532,40.942,61.285,-151.2010,26.0821,0.0000
C00841=-46.550,43.085,61.257,-153.0602,29.1088,0.0000
C00842=-44.848,44.848,61.276,-151.9510,28.0490,0.0000
C00843=-43.085,46.550,61.257,-150.8912,26.9398,0.0000
C00844=-40.942,48.532,61.285,-153.9179,28.7990,0.0000
C00845=-39.035,51.313,61.945,-176.2538,25.2815,0.0000
C00846=-39.736,54.260,63.612,179.8739,0.2177,0.0000
C00847=-42.239,58.063,65.929,-177.6803,-3.4830,0.0000
C00848=-45.816,62.906,68.324,-176.4893,-5.0463,0.0000
C00849=-49.842,68.316,70.157,-175.7728,-6.1010,0.0000
C00850=-53.356,73.536,71.060,-176.9924,-6.7977,0.0000
C00851=-54.130,79.138,71.535,179.3160,-4.6290,0.0000
C00852=-51.936,84.362,71.920,178.6069,-1.8286,0.0000
C00853=-47.191,88.127,72.309,179.8682,-0.0745,0.0000
C00854=-41.335,91.053,72.565,179.9828,-0.0057,0.0000
C00855=-35.156,93.612,72.565,179.9828,-0.0057,0.0000
C00856=-28.946,95.684,72.309,179.8568,-0.0401,0.0000
C00857=-22.929,96.378,71.920,177.7247,0.3096,0.0000
C00858=-17.683,94.235,71.535,176.2458,2.7916,0.0000
C00859=-14.270,89.726,71.060,177.2978,6.9230,0.0000
C00860=-13.063,83.550,70.157,178.6599,7.2864,0.0000
C00861=-12.084,76.878,68.324,178.9053,6.0453,0.0000
C00862=-11.189,70.924,65.929,179.1728,4.1007,0.0000
C00863=-10.270,66.465,63.612,-179.9370,-0.2406,0.0000
C00864=-8.682,63.886,61.945,-159.1815,-16.0518,0.0000
C00865=-5.367,63.268,61.285,-143.6885,-2.4389,0.0000
C00866=-2.450,63.381,61.257,-143.0189,1.9725,0.0000
C00867=0.000,63.425,61.276,-142.9995,-0.0000,0.0000
C00868=0.000,62.111,63.041,-143.6744,-0.0000,0.0000
C00869=2.330,62.072,63.021,-143.6941,-1.8769,0.0000
C00870=5.165,61.970,63.050,-144.4283,2.7471,0.0000
C00871=8.436,62.639,63.741,-160.6277,15.7061,0.0000
C00872=9.975,65.350,65.485,179.9141,-0.3495,0.0000
C00873=10.861,70.011,67.904,179.1957,-4.2040,0.0000
C00874=11.743,76.212,70.393,178.9746,-5.9073,0.0000
C00875=12.712,83.133,72.289,178.7761,-7.0035,0.0000
C00876=13.898,89.524,73.219,177.5072,-6.6505,0.0000
C00877=17.338,94.193,73.707,176.4297,-2.7222,0.0000
C00878=22.659,96.427,74.103,177.8280,-0.3096,0.0000
C00879=28.778,95.739,74.502,179.8625,0.0401,0.0000
C00880=35.099,93.634,74.765,179.9828,0.0057,0.0000
C00881=41.391,91.028,74.765,179.9828,0.0057,0.0000
C00882=47.349,88.047,74.502,179.8739,0.0688,0.0000
C00883=52.162,84.206,74.103,178.6815,1.7539,0.0000
C00884=54.344,78.865,73.707,179.3965,4.4453,0.0000
C00885=53.475,73.130,73.219,-177.0463,6.4568,0.0000
C00886=49.795,67.773,72.289,-175.8959,5.8232,0.0000
C00887=45.586,62.194,70.393,-176.5359,4.9024,0.0000
C00888=41.825,57.185,67.904,-177.5940,3.5463,0.0000
C00889=39.156,53.262,65.485,-179.8167,0.3094,0.0000
C00890=38.328,50.258,63.741,-177.1495,-24.1122,0.0000
C00891=40.167,47.472,63.050,-154.7409,-28.3520,0.0000
C00892=42.244,45.539,63.021,-151.5113,-26.3998,0.0000
C00893=43.919,43.919,63.041,-152.5292,-27.4708,0.0000
C00894=45.539,42.244,63.021,-153.6002,-28.4887,0.0000
C00895=47.472,40.167,63.050,-151.6480,-25.2534,0.0000
C00896=50.258,38.328,63.741,-155.8878,-2.8505,0.0000
C00897=53.262,39.156,65.485,179.6906,-0.1833,0.0000
C00898=57.185,41.825,67.904,176.4537,-2.4060,0.0000
C00899=62.194,45.586,70.393,175.0976,-3.4641,0.0000
C00900=67.773,49.795,72.289,174.1768,-4.1041,0.0000
C00901=73.130,53.475,73.219,173.5432,-2.9537,0.0000
C00902=78.865,54.344,73.707,175.5547,0.6035,0.0000
C00903=84.206,52.162,74.103,178.2461,1.3185,0.0000
C00904=88.047,47.349,74.502,179.9312,0.1261,0.0000
C00905=91.028,41.391,74.765,179.9943,0.0172,0.0000
C00906=93.634,35.099,74.765,179.9943,0.0172,0.0000
C00907=95.739,28.778,74.502,179.9599,0.1375,0.0000
C00908=96.427,22.659,74.103,-179.6904,2.1720,0.0000
C00909=94.193,17.338,73.707,-177.2778,3.5703,0.0000
C00910=89.524,13.898,73.219,-173.3495,2.4928,0.0000
C00911=83.133,12.712,72.289,-172.9965,1.2239,0.0000
C00912=76.212,11.743,70.393,-174.0927,1.0254,0.0000
C00913=70.011,10.861,67.904,-175.7960,0.8043,0.0000
C00914=65.350,9.975,65.485,-179.6505,0.0859,0.0000
C00915=62.639,8.436,63.741,164.2939,-19.3723,0.0000
C00916=61.970,5.165,63.050,177.2529,-35.5717,0.0000
C00917=62.072,2.330,63.021,-178.1231,-36.3059,0.0000
C00918=62.111,0.000,63.041,-180.0000,-36.3256,0.0000
C00919=62.072,-2.330,63.021,178.1231,-36.3059,0.0000
C00920=61.970,-5.165,63.050,-177.2529,-35.5717,0.0000
C00921=62.640,-8.436,63.741,-164.2939,-19.3723,0.0000
C00922=65.350,-9.975,65.485,179.6505,0.0859,0.0000
C00923=70.011,-10.861,67.904,175.7960,0.8043,0.0000
C00924=76.212,-11.743,70.393,174.0927,1.0254,0.0000
C00925=83.133,-12.712,72.289,172.9965,1.2239,0.0000
C00926=89.524,-13.898,73.219,173.3495,2.4928,0.0000
C00927=94.193,-17.338,73.707,177.2778,3.5703,0.0000
C00928=96.427,-22.659,74.103,179.6904,2.1720,0.0000
C00929=95.739,-28.778,74.502,-179.9599,0.1375,0.0000
C00930=93.634,-35.099,74.765,-179.9943,0.0172,0.0000
C00931=91.028,-41.391,74.765,-179.9943,0.0172,0.0000
C00932=88.047,-47.349,74.502,-179.9312,0.1261,0.0000
C00933=84.206,-52.162,74.103,-178.2461,1.3185,0.0000
C00934=78.865,-54.344,73.707,-175.5547,0.6035,0.0000
C00935=73.130,-53.475,73.219,-173.5432,-2.9537,0.0000
C00936=67.773,-49.795,72.289,-174.1768,-4.1041,0.0000
C00937=62.194,-45.586,70.393,-175.0976,-3.4641,0.0000
C00938=57.185,-41.825,67.904,-176.4537,-2.4060,0.0000
C00939=53.262,-39.156,65.485,-179.6906,-0.1833,0.0000
C00940=50.258,-38.328,63.741,155.8878,-2.8505,0.0000
C00941=47.472,-40.167,63.050,151.6480,-25.2591,0.0000
C00942=45.539,-42.244,63.021,153.6002,-28.4887,0.0000
C00943=43.919,-43.919,63.041,152.5292,-27.4708,0.0000
C00944=42.244,-45.539,63.021,151.5113,-26.3998,0.0000
C00945=40.167,-47.472,63.050,154.7466,-28.3520,0.0000
C00946=38.328,-50.258,63.741,177.1495,-24.1122,0.0000
C00947=39.156,-53.262,65.485,179.8167,0.3094,0.0000
C00948=41.825,-57.185,67.904,177.5940,3.5463,0.0000
C00949=45.586,-62.194,70.393,176.5359,4.9024,0.0000
C00950=49.795,-67.773,72.289,175.8959,5.8232,0.0000
C00951=53.475,-73.130,73.219,177.0463,6.4568,0.0000
C00952=54.344,-78.865,73.707,-179.3965,4.4453,0.0000
C00953=52.162,-84.206,74.103,-178.6815,1.7539,0.0000
C00954=47.349,-88.047,74.502,-179.8739,0.0688,0.0000
C00955=41.391,-91.028,74.765,-179.9828,0.0057,0.0000
C00956=35.099,-93.634,74.765,-179.9828,0.0057,0.0000
C00957=28.778,-95.739,74.502,-179.8625,0.0401,0.0000
C00958=22.659,-96.427,74.103,-177.8280,-0.3096,0.0000
C00959=17.338,-94.193,73.707,-176.4297,-2.7222,0.0000
C00960=13.898,-89.524,73.219,-177.5072,-6.6505,0.0000
C00961=12.712,-83.133,72.289,-178.7761,-7.0035,0.0000
C00962=11.743,-76.212,70.393,-178.9746,-5.9073,0.0000
C00963=10.861,-70.011,67.904,-179.1957,-4.2040,0.0000
C00964=9.975,-65.350,65.485,-179.9141,-0.3495,0.0000
C00965=8.436,-62.639,63.741,160.6277,15.7061,0.0000
C00966=5.165,-61.970,63.050,144.4283,2.7471,0.0000
C00967=2.330,-62.072,63.021,143.6941,-1.8769,0.0000
C00968=0.000,-62.111,63.041,143.6744,-0.0000,0.0000
C00969=0.000,-62.111,63.041,143.6744,-0.0000,0.0000
C00970=-2.330,-62.072,63.021,143.6941,1.8769,0.0000
C00971=-5.165,-61.970,63.050,144.4283,-2.7471,0.0000
C00972=-8.436,-62.640,63.741,160.6277,-15.7061,0.0000
C00973=-9.975,-65.350,65.485,-179.9141,0.3495,0.0000
C00974=-10.861,-70.011,67.904,-179.1957,4.2040,0.0000
C00975=-11.743,-76.212,70.393,-178.9746,5.9073,0.0000
C00976=-12.712,-83.133,72.289,-178.7761,7.0035,0.0000
C00977=-13.898,-89.524,73.219,-177.5072,6.6505,0.0000
C00978=-17.338,-94.193,73.707,-176.4297,2.7222,0.0000
C00979=-22.659,-96.427,74.103,-177.8280,0.3096,0.0000
C00980=-28.778,-95.739,74.502,-179.8625,-0.0401,0.0000
C00981=-35.099,-93.634,74.765,-179.9828,-0.0057,0.0000
C00982=-41.391,-91.028,74.765,-179.9828,-0.0057,0.0000
C00983=-47.349,-88.047,74.502,-179.8739,-0.0688,0.0000
C00984=-52.162,-84.206,74.103,-178.6815,-1.7539,0.0000
C00985=-54.344,-78.865,73.707,-179.3965,-4.4453,0.0000
C00986=-53.475,-73.130,73.219,177.0463,-6.4568,0.0000
C00987=-49.795,-67.773,72.289,175.8959,-5.8232,0.0000
C00988=-45.586,-62.194,70.393,176.5359,-4.9024,0.0000
C00989=-41.825,-57.185,67.904,177.5940,-3.5463,0.0000
C00990=-39.156,-53.262,65.485,179.8167,-0.3094,0.0000
C00991=-38.328,-50.258,63.741,177.1495,24.1122,0.0000
C00992=-40.167,-47.472,63.050,154.7409,28.3520,0.0000
C00993=-42.244,-45.539,63.021,151.5113,26.3998,0.0000
C00994=-43.919,-43.919,63.041,152.5292,27.4708,0.0000
C00995=-45.539,-42.244,63.021,153.6002,28.4887,0.0000
C00996=-47.472,-40.167,63.050,151.6480,25.2534,0.0000
C00997=-50.258,-38.328,63.741,155.8878,2.8505,0.0000
C00998=-53.262,-39.156,65.485,-179.6906,0.1833,0.0000
C00999=-57.185,-41.825,67.904,-176.4537,2.4060,0.0000
C01000=-62.194,-45.586,70.393,-175.0976,3.4641,0.0000
C01001=-67.773,-49.795,72.289,-174.1768,4.1041,0.0000
C01002=-73.130,-53.475,73.219,-173.5432,2.9537,0.0000
C01003=-78.865,-54.344,73.707,-175.5547,-0.6035,0.0000
C01004=-84.206,-52.162,74.103,-178.2461,-1.3185,0.0000
C01005=-88.047,-47.349,74.502,-179.9312,-0.1261,0.0000
C01006=-91.028,-41.391,74.765,-179.9943,-0.0172,0.0000
C01007=-93.634,-35.099,74.765,-179.9943,-0.0172,0.0000
C01008=-95.739,-28.778,74.502,-179.9599,-0.1375,0.0000
C01009=-96.427,-22.659,74.103,179.6904,-2.1720,0.0000
C01010=-94.193,-17.338,73.707,177.2778,-3.5703,0.0000
C01011=-89.524,-13.898,73.219,173.3495,-2.4928,0.0000
C01012=-83.133,-12.712,72.289,172.9965,-1.2239,0.0000
C01013=-76.212,-11.743,70.393,174.0927,-1.0254,0.0000
C01014=-70.011,-10.861,67.904,175.7960,-0.8043,0.0000
C01015=-65.350,-9.975,65.485,179.6505,-0.0859,0.0000
C01016=-62.639,-8.436,63.741,-164.2939,19.3723,0.0000
C01017=-61.970,-5.165,63.050,-177.2529,35.5717,0.0000
C01018=-62.072,-2.330,63.021,178.1231,36.3059,0.0000
C01019=-62.111,0.000,63.041,180.0000,36.3256,0.0000
C01020=-62.072,2.330,63.021,-178.1231,36.3059,0.0000
C01021=-61.970,5.165,63.050,177.2529,35.5717,0.0000
C01022=-62.640,8.436,63.741,164.2939,19.3723,0.0000
C01023=-65.350,9.975,65.485,-179.6505,-0.0859,0.0000
C01024=-70.011,10.861,67.904,-175.7960,-0.8043,0.0000
C01025=-76.212,11.743,70.393,-174.0927,-1.0254,0.0000
C01026=-83.133,12.712,72.289,-172.9965,-1.2239,0.0000
C01027=-89.524,13.898,73.219,-173.3495,-2.4928,0.0000
C01028=-94.193,17.338,73.707,-177.2778,-3.5703,0.0000
C01029=-96.427,22.659,74.103,-179.6904,-2.1720,0.0000
C01030=-95.739,28.778,74.502,179.9599,-0.1375,0.0000
C01031=-93.634,35.099,74.765,179.9943,-0.0172,0.0000
C01032=-91.028,41.391,74.765,179.9943,-0.0172,0.0000
C01033=-88.047,47.349,74.502,179.9312,-0.1261,0.0000
C01034=-84.206,52.162,74.103,178.2461,-1.3185,0.0000
C01035=-78.865,54.344,73.707,175.5547,-0.6035,0.0000
C01036=-73.130,53.475,73.219,173.5432,2.9537,0.0000
C01037=-67.773,49.795,72.289,174.1768,4.1041,0.0000
C01038=-62.194,45.586,70.393,175.0976,3.4641,0.0000
C01039=-57.185,41.825,67.904,176.4537,2.4060,0.0000
C01040=-53.262,39.156,65.485,179.6906,0.1833,0.0000
C01041=-50.258,38.328,63.741,-155.8878,2.8505,0.0000
C01042=-47.472,40.167,63.050,-151.6480,25.2591,0.0000
C01043=-45.539,42.244,63.021,-153.6002,28.4887,0.0000
C01044=-43.919,43.919,63.041,-152.5292,27.4708,0.0000
C01045=-42.244,45.539,63.021,-151.5113,26.3998,0.0000
C01046=-40.167,47.472,63.050,-154.7466,28.3520,0.0000
C01047=-38.328,50.258,63.741,-177.1495,24.1122,0.0000
C01048=-39.156,53.262,65.485,-179.8167,-0.3094,0.0000
C01049=-41.825,57.185,67.904,-177.5940,-3.5463,0.0000
C01050=-45.586,62.194,70.393,-176.5359,-4.9024,0.0000
C01051=-49.795,67.773,72.289,-175.8959,-5.8232,0.0000
C01052=-53.475,73.130,73.219,-177.0463,-6.4568,0.0000
C01053=-54.344,78.865,73.707,179.3965,-4.4453,0.0000
C01054=-52.162,84.206,74.103,178.6815,-1.7539,0.0000
C01055=-47.349,88.047,74.502,179.8739,-0.0688,0.0000
C01056=-41.391,91.028,74.765,179.9828,-0.0057,0.0000
C01057=-35.099,93.634,74.765,179.9828,-0.0057,0.0000
C01058=-28.778,95.739,74.502,179.8625,-0.0401,0.0000
C01059=-22.659,96.427,74.103,177.8280,0.3096,0.0000
C01060=-17.338,94.193,73.707,176.4297,2.7222,0.0000
C01061=-13.898,89.524,73.219,177.5072,6.6505,0.0000
C01062=-12.712,83.133,72.289,178.7761,7.0035,0.0000
C01063=-11.743,76.212,70.393,178.9746,5.9073,0.0000
C01064=-10.861,70.011,67.904,179.1957,4.2040,0.0000
C01065=-9.975,65.350,65.485,179.9141,0.3495,0.0000
C01066=-8.436,62.640,63.741,-160.6277,-15.7061,0.0000
C01067=-5.165,61.970,63.050,-144.4283,-2.7471,0.0000
C01068=-2.330,62.072,63.021,-143.6941,1.8769,0.0000
C01069=0.000,62.111,63.041,-143.6744,-0.0000,0.0000
C01070=0.000,60.820,64.822,-144.4503,-0.0000,0.0000
C01071=2.212,60.785,64.801,-144.4657,-1.7813,0.0000
C01072=4.967,60.695,64.832,-145.2744,3.0326,0.0000
C01073=8.195,61.417,65.554,-162.0686,15.2578,0.0000
C01074=9.686,64.262,67.375,179.7994,-0.8537,0.0000
C01075=10.544,69.129,69.894,179.2244,-4.2440,0.0000
C01076=11.418,75.576,72.474,179.0499,-5.7112,0.0000
C01077=12.382,82.740,74.428,178.8866,-6.6509,0.0000
C01078=13.550,89.334,75.383,177.7168,-6.3028,0.0000
C01079=17.016,94.154,75.883,176.6487,-2.6122,0.0000
C01080=22.407,96.473,76.288,177.9483,-0.3039,0.0000
C01081=28.621,95.791,76.696,179.8682,0.0401,0.0000
C01082=35.046,93.654,76.964,179.9828,0.0057,0.0000
C01083=41.442,91.005,76.964,179.9828,0.0057,0.0000
C01084=47.497,87.973,76.696,179.8797,0.0630,0.0000
C01085=52.372,84.060,76.288,178.7675,1.6623,0.0000
C01086=54.545,78.609,75.883,179.4772,4.2093,0.0000
C01087=53.588,72.750,75.383,-177.1410,6.0691,0.0000
C01088=49.751,67.261,74.428,-176.0657,5.4929,0.0000
C01089=45.367,61.514,72.474,-176.6234,4.7117,0.0000
C01090=41.426,56.337,69.894,-177.5424,3.5520,0.0000
C01091=38.591,52.289,67.375,-179.5416,0.7449,0.0000
C01092=37.634,49.223,65.554,-177.9415,-22.8629,0.0000
C01093=39.406,46.429,64.832,-155.6444,-27.8155,0.0000
C01094=41.417,44.545,64.801,-152.2116,-25.7851,0.0000
C01095=43.006,43.006,64.822,-153.1932,-26.8068,0.0000
C01096=44.545,41.417,64.801,-154.2149,-27.7884,0.0000
C01097=46.430,39.405,64.832,-152.1845,-24.3498,0.0000
C01098=49.223,37.634,65.554,-157.1371,-2.0585,0.0000
C01099=52.289,38.591,67.375,179.2551,-0.4584,0.0000
C01100=56.337,41.426,69.894,176.4480,-2.4576,0.0000
C01101=61.514,45.367,72.474,175.2883,-3.3766,0.0000
C01102=67.261,49.751,74.428,174.5071,-3.9343,0.0000
C01103=72.750,53.588,75.383,173.9309,-2.8590,0.0000
C01104=78.609,54.545,75.883,175.7907,0.5228,0.0000
C01105=84.060,52.372,76.288,178.3377,1.2325,0.0000
C01106=87.973,47.497,76.696,179.9370,0.1203,0.0000
C01107=91.005,41.442,76.964,179.9943,0.0172,0.0000
C01108=93.654,35.046,76.964,179.9943,0.0172,0.0000
C01109=95.791,28.621,76.696,179.9599,0.1318,0.0000
C01110=96.473,22.407,76.288,-179.6961,2.0517,0.0000
C01111=94.154,17.016,75.883,-177.3878,3.3513,0.0000
C01112=89.334,13.550,75.383,-173.6972,2.2832,0.0000
C01113=82.740,12.382,74.428,-173.3491,1.1134,0.0000
C01114=75.576,11.418,72.474,-174.2888,0.9501,0.0000
C01115=69.129,10.544,69.894,-175.7560,0.7756,0.0000
C01116=64.262,9.686,67.375,-179.1463,0.2006,0.0000
C01117=61.417,8.195,65.554,164.7422,-17.9314,0.0000
C01118=60.695,4.967,64.832,176.9674,-34.7256,0.0000
C01119=60.785,2.212,64.801,-178.2187,-35.5343,0.0000
C01120=60.820,0.000,64.822,-180.0000,-35.5497,0.0000
C01121=60.785,-2.212,64.801,178.2187,-35.5343,0.0000
C01122=60.695,-4.967,64.832,-176.9674,-34.7256,0.0000
C01123=61.417,-8.195,65.554,-164.7422,-17.9314,0.0000
C01124=64.262,-9.686,67.375,179.1463,0.2006,0.0000
C01125=69.129,-10.544,69.894,175.7560,0.7756,0.0000
C01126=75.576,-11.418,72.474,174.2888,0.9501,0.0000
C01127=82.740,-12.382,74.428,173.3491,1.1134,0.0000
C01128=89.334,-13.550,75.383,173.6972,2.2832,0.0000
C01129=94.154,-17.016,75.883,177.3878,3.3513,0.0000
C01130=96.473,-22.407,76.288,179.6961,2.0517,0.0000
C01131=95.791,-28.621,76.696,-179.9599,0.1318,0.0000
C01132=93.654,-35.046,76.964,-179.9943,0.0172,0.0000
C01133=91.005,-41.442,76.964,-179.9943,0.0172,0.0000
C01134=87.973,-47.497,76.696,-179.9370,0.1203,0.0000
C01135=84.060,-52.372,76.288,-178.3377,1.2325,0.0000
C01136=78.609,-54.545,75.883,-175.7907,0.5228,0.0000
C01137=72.750,-53.588,75.383,-173.9309,-2.8590,0.0000
C01138=67.261,-49.751,74.428,-174.5071,-3.9343,0.0000
C01139=61.514,-45.367,72.474,-175.2883,-3.3766,0.0000
C01140=56.337,-41.426,69.894,-176.4480,-2.4576,0.0000
C01141=52.289,-38.591,67.375,-179.2551,-0.4584,0.0000
C01142=49.223,-37.634,65.554,157.1371,-2.0585,0.0000
C01143=46.429,-39.406,64.832,152.1845,-24.3556,0.0000
C01144=44.545,-41.417,64.801,154.2149,-27.7884,0.0000
C01145=43.006,-43.006,64.822,153.1932,-26.8068,0.0000
C01146=41.417,-44.545,64.801,152.2116,-25.7851,0.0000
C01147=39.405,-46.430,64.832,155.6502,-27.8155,0.0000
C01148=37.634,-49.223,65.554,177.9415,-22.8629,0.0000
C01149=38.591,-52.289,67.375,179.5416,0.7449,0.0000
C01150=41.426,-56.337,69.894,177.5424,3.5520,0.0000
C01151=45.367,-61.514,72.474,176.6234,4.7117,0.0000
C01152=49.751,-67.261,74.428,176.0657,5.4929,0.0000
C01153=53.588,-72.750,75.383,177.1410,6.0691,0.0000
C01154=54.545,-78.609,75.883,-179.4772,4.2093,0.0000
C01155=52.372,-84.060,76.288,-178.7675,1.6623,0.0000
C01156=47.497,-87.973,76.696,-179.8797,0.0630,0.0000
C01157=41.442,-91.005,76.964,-179.9828,0.0057,0.0000
C01158=35.046,-93.654,76.964,-179.9828,0.0057,0.0000
C01159=28.621,-95.791,76.696,-179.8682,0.0401,0.0000
C01160=22.407,-96.473,76.288,-177.9483,-0.3039,0.0000
C01161=17.016,-94.154,75.883,-176.6487,-2.6122,0.0000
C01162=13.550,-89.334,75.383,-177.7168,-6.3028,0.0000
C01163=12.382,-82.740,74.428,-178.8866,-6.6509,0.0000
C01164=11.418,-75.576,72.474,-179.0499,-5.7112,0.0000
C01165=10.544,-69.129,69.894,-179.2244,-4.2440,0.0000
C01166=9.686,-64.262,67.375,-179.7994,-0.8537,0.0000
C01167=8.195,-61.417,65.554,162.0686,15.2578,0.0000
C01168=4.967,-60.695,64.832,145.2744,3.0326,0.0000
C01169=2.212,-60.785,64.801,144.4657,-1.7813,0.0000
C01170=0.000,-60.820,64.822,144.4503,-0.0000,0.0000
C01171=0.000,-60.820,64.822,144.4503,-0.0000,0.0000
C01172=-2.212,-60.785,64.801,144.4657,1.7813,0.0000
C01173=-4.967,-60.695,64.832,145.2744,-3.0326,0.0000
C01174=-8.195,-61.417,65.554,162.0686,-15.2578,0.0000
C01175=-9.686,-64.262,67.375,-179.7994,0.8537,0.0000
C01176=-10.544,-69.129,69.894,-179.2244,4.2440,0.0000
C01177=-11.418,-75.576,72.474,-179.0499,5.7112,0.0000
C01178=-12.382,-82.740,74.428,-178.8866,6.6509,0.0000
C01179=-13.550,-89.334,75.383,-177.7168,6.3028,0.0000
C01180=-17.016,-94.154,75.883,-176.6487,2.6122,0.0000
C01181=-22.407,-96.473,76.288,-177.9483,0.3039,0.0000
C01182=-28.621,-95.791,76.696,-179.8682,-0.0401,0.0000
C01183=-35.046,-93.654,76.964,-179.9828,-0.0057,0.0000
C01184=-41.442,-91.005,76.964,-179.9828,-0.0057,0.0000
C01185=-47.497,-87.973,76.696,-179.8797,-0.0630,0.0000
C01186=-52.372,-84.060,76.288,-178.7675,-1.6623,0.0000
C01187=-54.545,-78.609,75.883,-179.4772,-4.2093,0.0000
C01188=-53.588,-72.750,75.383,177.1410,-6.0691,0.0000
C01189=-49.751,-67.261,74.428,176.0657,-5.4929,0.0000
C01190=-45.367,-61.514,72.474,176.6234,-4.7117,0.0000
C01191=-41.426,-56.337,69.894,177.5424,-3.5520,0.0000
C01192=-38.591,-52.289,67.375,179.5416,-0.7449,0.0000
C01193=-37.634,-49.223,65.554,177.9415,22.8629,0.0000
C01194=-39.406,-46.429,64.832,155.6444,27.8155,0.0000
C01195=-41.417,-44.545,64.801,152.2116,25.7851,0.0000
C01196=-43.006,-43.006,64.822,153.1932,26.8068,0.0000
C01197=-44.545,-41.417,64.801,154.2149,27.7884,0.0000
C01198=-46.430,-39.405,64.832,152.1845,24.3498,0.0000
C01199=-49.223,-37.634,65.554,157.1371,2.0585,0.0000
C01200=-52.289,-38.591,67.375,-179.2551,0.4584,0.0000
C01201=-56.337,-41.426,69.894,-176.4480,2.4576,0.0000
C01202=-61.514,-45.367,72.474,-175.2883,3.3766,0.0000
C01203=-67.261,-49.751,74.428,-174.5071,3.9343,0.0000
C01204=-72.750,-53.588,75.383,-173.9309,2.8590,0.0000
C01205=-78.609,-54.545,75.883,-175.7907,-0.5228,0.0000
C01206=-84.060,-52.372,76.288,-178.3377,-1.2325,0.0000
C01207=-87.973,-47.497,76.696,-179.9370,-0.1203,0.0000
C01208=-91.005,-41.442,76.964,-179.9943,-0.0172,0.0000
C01209=-93.654,-35.046,76.964,-179.9943,-0.0172,0.0000
C01210=-95.791,-28.621,76.696,-179.9599,-0.1318,0.0000
C01211=-96.473,-22.407,76.288,179.6961,-2.0517,0.0000
C01212=-94.154,-17.016,75.883,177.3878,-3.3513,0.0000
C01213=-89.334,-13.550,75.383,173.6972,-2.2832,0.0000
C01214=-82.740,-12.382,74.428,173.3491,-1.1134,0.0000
C01215=-75.576,-11.418,72.474,174.2888,-0.9501,0.0000
C01216=-69.129,-10.544,69.894,175.7560,-0.7756,0.0000
C01217=-64.262,-9.686,67.375,179.1463,-0.2006,0.0000
C01218=-61.417,-8.195,65.554,-164.7422,17.9314,0.0000
C01219=-60.695,-4.967,64.832,-176.9674,34.7256,0.0000
C01220=-60.785,-2.212,64.801,178.2187,35.5343,0.0000
C01221=-60.820,0.000,64.822,180.0000,35.5497,0.0000
C01222=-60.785,2.212,64.801,-178.2187,35.5343,0.0000
C01223=-60.695,4.967,64.832,176.9674,34.7256,0.0000
C01224=-61.417,8.195,65.554,164.7422,17.9314,0.0000
C01225=-64.262,9.686,67.375,-179.1463,-0.2006,0.0000
C01226=-69.129,10.544,69.894,-175.7560,-0.7756,0.0000
C01227=-75.576,11.418,72.474,-174.2888,-0.9501,0.0000
C01228=-82.740,12.382,74.428,-173.3491,-1.1134,0.0000
C01229=-89.334,13.550,75.383,-173.6972,-2.2832,0.0000
C01230=-94.154,17.016,75.883,-177.3878,-3.3513,0.0000
C01231=-96.473,22.407,76.288,-179.6961,-2.0517,0.0000
C01232=-95.791,28.621,76.696,179.9599,-0.1318,0.0000
C01233=-93.654,35.046,76.964,179.9943,-0.0172,0.0000
C01234=-91.005,41.442,76.964,179.9943,-0.0172,0.0000
C01235=-87.973,47.497,76.696,179.9370,-0.1203,0.0000
C01236=-84.060,52.372,76.288,178.3377,-1.2325,0.0000
C01237=-78.609,54.545,75.883,175.7907,-0.5228,0.0000
C01238=-72.750,53.588,75.383,173.9309,2.8590,0.0000
C01239=-67.261,49.751,74.428,174.5071,3.9343,0.0000
C01240=-61.514,45.367,72.474,175.2883,3.3766,0.0000
C01241=-56.337,41.426,69.894,176.4480,2.4576,0.0000
C01242=-52.289,38.591,67.375,179.2551,0.4584,0.0000
C01243=-49.223,37.634,65.554,-157.1371,2.0585,0.0000
C01244=-46.429,39.406,64.832,-152.1845,24.3556,0.0000
C01245=-44.545,41.417,64.801,-154.2149,27.7884,0.0000
C01246=-43.006,43.006,64.822,-153.1932,26.8068,0.0000
C01247=-41.417,44.545,64.801,-152.2116,25.7851,0.0000
C01248=-39.405,46.430,64.832,-155.6502,27.8155,0.0000
C01249=-37.634,49.223,65.554,-177.9415,22.8629,0.0000
C01250=-38.591,52.289,67.375,-179.5416,-0.7449,0.0000
C01251=-41.426,56.337,69.894,-177.5424,-3.5520,0.0000
C01252=-45.367,61.514,72.474,-176.6234,-4.7117,0.0000
C01253=-49.751,67.261,74.428,-176.0657,-5.4929,0.0000
C01254=-53.588,72.750,75.383,-177.1410,-6.0691,0.0000
C01255=-54.545,78.609,75.883,179.4772,-4.2093,0.0000
C01256=-52.372,84.060,76.288,178.7675,-1.6623,0.0000
C01257=-47.497,87.973,76.696,179.8797,-0.0630,0.0000
C01258=-41.442,91.005,76.964,179.9828,-0.0057,0.0000
C01259=-35.046,93.654,76.964,179.9828,-0.0057,0.0000
C01260=-28.621,95.791,76.696,179.8682,-0.0401,0.0000
C01261=-22.407,96.473,76.288,177.9483,0.3039,0.0000
C01262=-17.016,94.154,75.883,176.6487,2.6122,0.0000
C01263=-13.550,89.334,75.383,177.7168,6.3028,0.0000
C01264=-12.382,82.740,74.428,178.8866,6.6509,0.0000
C01265=-11.418,75.576,72.474,179.0499,5.7112,0.0000
C01266=-10.544,69.129,69.894,179.2244,4.2440,0.0000
C01267=-9.686,64.262,67.375,179.7994,0.8537,0.0000
C01268=-8.195,61.417,65.554,-162.0686,-15.2578,0.0000
C01269=-4.967,60.695,64.832,-145.2744,-3.0326,0.0000
C01270=-2.212,60.785,64.801,-144.4657,1.7813,0.0000
C01271=0.000,60.820,64.822,-144.4503,-0.0000,0.0000
C01272=0.000,59.554,66.621,-145.3422,-0.0000,0.0000
C01273=2.097,59.523,66.599,-145.3578,-1.6714,0.0000
C01274=4.772,59.445,66.632,-146.2336,3.2876,0.0000
C01275=7.959,60.221,67.386,-163.5011,14.7099,0.0000
C01276=9.406,63.206,69.285,179.7192,-1.2721,0.0000
C01277=10.239,68.282,71.901,179.2646,-4.2269,0.0000
C01278=11.109,74.974,74.567,179.1251,-5.4574,0.0000
C01279=12.073,82.372,76.575,179.0028,-6.2415,0.0000
C01280=13.226,89.158,77.551,177.9318,-5.8869,0.0000
C01281=16.717,94.118,78.062,176.9016,-2.4681,0.0000
C01282=22.174,96.515,78.476,178.0973,-0.2924,0.0000
C01283=28.477,95.839,78.891,179.8797,0.0344,0.0000
C01284=34.998,93.673,79.163,179.9885,0.0057,0.0000
C01285=41.489,90.984,79.163,179.9885,0.0057,0.0000
C01286=47.632,87.904,78.891,179.8911,0.0630,0.0000
C01287=52.567,83.926,78.476,178.8593,1.5533,0.0000
C01288=54.731,78.373,78.062,179.5520,3.9338,0.0000
C01289=53.692,72.396,77.551,-177.2816,5.6244,0.0000
C01290=49.709,66.782,76.575,-176.2812,5.1227,0.0000
C01291=45.159,60.870,74.567,-176.7513,4.4806,0.0000
C01292=41.042,55.523,71.901,-177.5309,3.5119,0.0000
C01293=38.042,51.344,69.285,-179.3008,1.1003,0.0000
C01294=36.955,48.211,67.386,-178.6323,-21.5556,0.0000
C01295=38.660,45.408,66.632,-156.6317,-27.1745,0.0000
C01296=40.607,43.572,66.599,-153.0157,-25.0779,0.0000
C01297=42.111,42.111,66.621,-153.9499,-26.0501,0.0000
C01298=43.571,40.607,66.599,-154.9221,-26.9898,0.0000
C01299=45.409,38.659,66.632,-152.8255,-23.3683,0.0000
C01300=48.211,36.955,67.386,-158.4444,-1.3616,0.0000
C01301=51.344,38.042,69.285,178.8997,-0.6992,0.0000
C01302=55.523,41.042,71.901,176.4881,-2.4691,0.0000
C01303=60.870,45.159,74.567,175.5194,-3.2487,0.0000
C01304=66.782,49.709,76.575,174.8773,-3.7188,0.0000
C01305=72.396,53.692,77.551,174.3756,-2.7184,0.0000
C01306=78.373,54.731,78.062,176.0662,0.4480,0.0000
C01307=83.926,52.567,78.476,178.4467,1.1407,0.0000
C01308=87.904,47.632,78.891,179.9370,0.1089,0.0000
C01309=90.984,41.489,79.163,179.9943,0.0115,0.0000
C01310=93.673,34.998,79.163,179.9943,0.0115,0.0000
C01311=95.839,28.477,78.891,179.9656,0.1203,0.0000
C01312=96.515,22.174,78.476,-179.7076,1.9027,0.0000
C01313=94.118,16.717,78.062,-177.5319,3.0984,0.0000
C01314=89.158,13.226,77.551,-174.1131,2.0682,0.0000
C01315=82.372,12.073,76.575,-173.7585,0.9972,0.0000
C01316=74.974,11.109,74.567,-174.5426,0.8749,0.0000
C01317=68.282,10.239,71.901,-175.7731,0.7354,0.0000
C01318=63.206,9.406,69.285,-178.7279,0.2808,0.0000
C01319=60.221,7.959,67.386,165.2901,-16.4989,0.0000
C01320=59.445,4.772,66.632,176.7124,-33.7664,0.0000
C01321=59.523,2.097,66.599,-178.3286,-34.6422,0.0000
C01322=59.554,0.000,66.621,-180.0000,-34.6578,0.0000
C01323=59.523,-2.096,66.599,178.3286,-34.6422,0.0000
C01324=59.445,-4.772,66.632,-176.7124,-33.7617,0.0000
C01325=60.222,-7.959,67.386,-165.2901,-16.4989,0.0000
C01326=63.206,-9.406,69.285,178.7279,0.2808,0.0000
C01327=68.282,-10.239,71.901,175.7731,0.7354,0.0000
C01328=74.974,-11.109,74.567,174.5426,0.8749,0.0000
C01329=82.372,-12.073,76.575,173.7585,0.9972,0.0000
C01330=89.158,-13.226,77.551,174.1131,2.0682,0.0000
C01331=94.118,-16.717,78.062,177.5319,3.0984,0.0000
C01332=96.515,-22.174,78.476,179.7076,1.9027,0.0000
C01333=95.839,-28.477,78.891,-179.9656,0.1203,0.0000
C01334=93.673,-34.998,79.163,-179.9943,0.0115,0.0000
C01335=90.984,-41.489,79.163,-179.9943,0.0115,0.0000
C01336=87.904,-47.632,78.891,-179.9370,0.1089,0.0000
C01337=83.926,-52.567,78.476,-178.4467,1.1407,0.0000
C01338=78.373,-54.731,78.062,-176.0662,0.4480,0.0000
C01339=72.396,-53.692,77.551,-174.3756,-2.7184,0.0000
C01340=66.782,-49.709,76.575,-174.8773,-3.7188,0.0000
C01341=60.870,-45.159,74.567,-175.5194,-3.2487,0.0000
C01342=55.523,-41.042,71.901,-176.4881,-2.4691,0.0000
C01343=51.344,-38.042,69.285,-178.8997,-0.6992,0.0000
C01344=48.211,-36.955,67.386,158.4444,-1.3677,0.0000
C01345=45.408,-38.660,66.632,152.8255,-23.3683,0.0000
C01346=43.572,-40.607,66.599,154.9221,-26.9843,0.0000
C01347=42.111,-42.111,66.621,153.9499,-26.0501,0.0000
C01348=40.607,-43.571,66.599,153.0102,-25.0779,0.0000
C01349=38.659,-45.409,66.632,156.6317,-27.1745,0.0000
C01350=36.955,-48.211,67.386,178.6384,-21.5556,0.0000
C01351=38.042,-51.344,69.285,179.3008,1.1003,0.0000
C01352=41.042,-55.523,71.901,177.5309,3.5119,0.0000
C01353=45.159,-60.870,74.567,176.7513,4.4806,0.0000
C01354=49.709,-66.782,76.575,176.2812,5.1227,0.0000
C01355=53.692,-72.396,77.551,177.2816,5.6244,0.0000
C01356=54.731,-78.373,78.062,-179.5520,3.9338,0.0000
C01357=52.567,-83.926,78.476,-178.8593,1.5533,0.0000
C01358=47.632,-87.904,78.891,-179.8911,0.0630,0.0000
C01359=41.489,-90.984,79.163,-179.9885,0.0057,0.0000
C01360=34.998,-93.673,79.163,-179.9885,0.0057,0.0000
C01361=28.477,-95.839,78.891,-179.8797,0.0344,0.0000
C01362=22.174,-96.515,78.476,-178.0973,-0.2924,0.0000
C01363=16.717,-94.118,78.062,-176.9016,-2.4681,0.0000
C01364=13.226,-89.158,77.551,-177.9318,-5.8869,0.0000
C01365=12.073,-82.372,76.575,-179.0028,-6.2415,0.0000
C01366=11.109,-74.974,74.567,-179.1251,-5.4574,0.0000
C01367=10.239,-68.282,71.901,-179.2646,-4.2269,0.0000
C01368=9.406,-63.206,69.285,-179.7192,-1.2721,0.0000
C01369=7.959,-60.221,67.386,163.5011,14.7099,0.0000
C01370=4.772,-59.445,66.632,146.2336,3.2876,0.0000
C01371=2.097,-59.523,66.599,145.3578,-1.6714,0.0000
C01372=0.000,-59.554,66.621,145.3422,-0.0000,0.0000
C01373=0.000,-59.554,66.621,145.3422,-0.0000,0.0000
C01374=-2.096,-59.523,66.599,145.3578,1.6714,0.0000
C01375=-4.772,-59.445,66.632,146.2383,-3.2876,0.0000
C01376=-7.959,-60.222,67.386,163.5011,-14.7099,0.0000
C01377=-9.406,-63.206,69.285,-179.7192,1.2721,0.0000
C01378=-10.239,-68.282,71.901,-179.2646,4.2269,0.0000
C01379=-11.109,-74.974,74.567,-179.1251,5.4574,0.0000
C01380=-12.073,-82.372,76.575,-179.0028,6.2415,0.0000
C01381=-13.226,-89.158,77.551,-177.9318,5.8869,0.0000
C01382=-16.717,-94.118,78.062,-176.9016,2.4681,0.0000
C01383=-22.174,-96.515,78.476,-178.0973,0.2924,0.0000
C01384=-28.477,-95.839,78.891,-179.8797,-0.0344,0.0000
C01385=-34.998,-93.673,79.163,-179.9885,-0.0057,0.0000
C01386=-41.489,-90.984,79.163,-179.9885,-0.0057,0.0000
C01387=-47.632,-87.904,78.891,-179.8911,-0.0630,0.0000
C01388=-52.567,-83.926,78.476,-178.8593,-1.5533,0.0000
C01389=-54.731,-78.373,78.062,-179.5520,-3.9338,0.0000
C01390=-53.692,-72.396,77.551,177.2816,-5.6244,0.0000
C01391=-49.709,-66.782,76.575,176.2812,-5.1227,0.0000
C01392=-45.159,-60.870,74.567,176.7513,-4.4806,0.0000
C01393=-41.042,-55.523,71.901,177.5309,-3.5119,0.0000
C01394=-38.042,-51.344,69.285,179.3008,-1.1003,0.0000
C01395=-36.955,-48.211,67.386,178.6323,21.5556,0.0000
C01396=-38.660,-45.408,66.632,156.6317,27.1745,0.0000
C01397=-40.607,-43.572,66.599,153.0157,25.0779,0.0000
C01398=-42.111,-42.111,66.621,153.9499,26.0501,0.0000
C01399=-43.571,-40.607,66.599,154.9221,26.9898,0.0000
C01400=-45.409,-38.659,66.632,152.8255,23.3683,0.0000
C01401=-48.211,-36.955,67.386,158.4444,1.3616,0.0000
C01402=-51.344,-38.042,69.285,-178.8997,0.6992,0.0000
C01403=-55.523,-41.042,71.901,-176.4881,2.4691,0.0000
C01404=-60.870,-45.159,74.567,-175.5194,3.2487,0.0000
C01405=-66.782,-49.709,76.575,-174.8773,3.7188,0.0000
C01406=-72.396,-53.692,77.551,-174.3756,2.7184,0.0000
C01407=-78.373,-54.731,78.062,-176.0662,-0.4480,0.0000
C01408=-83.926,-52.567,78.476,-178.4467,-1.1407,0.0000
C01409=-87.904,-47.632,78.891,-179.9370,-0.1089,0.0000
C01410=-90.984,-41.489,79.163,-179.9943,-0.0115,0.0000
C01411=-93.673,-34.998,79.163,-179.9943,-0.0115,0.0000
C01412=-95.839,-28.477,78.891,-179.9656,-0.1203,0.0000
C01413=-96.515,-22.174,78.476,179.7076,-1.9027,0.0000
C01414=-94.118,-16.717,78.062,177.5319,-3.0984,0.0000
C01415=-89.158,-13.226,77.551,174.1131,-2.0682,0.0000
C01416=-82.372,-12.073,76.575,173.7585,-0.9972,0.0000
C01417=-74.974,-11.109,74.567,174.5426,-0.8749,0.0000
C01418=-68.282,-10.239,71.901,175.7731,-0.7354,0.0000
C01419=-63.206,-9.406,69.285,178.7279,-0.2808,0.0000
C01420=-60.221,-7.959,67.386,-165.2901,16.4989,0.0000
C01421=-59.445,-4.772,66.632,-176.7124,33.7664,0.0000
C01422=-59.523,-2.097,66.599,178.3286,34.6422,0.0000
C01423=-59.554,0.000,66.621,180.0000,34.6578,0.0000
C01424=-59.523,2.096,66.599,-178.3286,34.6422,0.0000
C01425=-59.445,4.772,66.632,176.7124,33.7617,0.0000
C01426=-60.222,7.959,67.386,165.2901,16.4989,0.0000
C01427=-63.206,9.406,69.285,-178.7279,-0.2808,0.0000
C01428=-68.282,10.239,71.901,-175.7731,-0.7354,0.0000
C01429=-74.974,11.109,74.567,-174.5426,-0.8749,0.0000
C01430=-82.372,12.073,76.575,-173.7585,-0.9972,0.0000
C01431=-89.158,13.226,77.551,-174.1131,-2.0682,0.0000
C01432=-94.118,16.717,78.062,-177.5319,-3.0984,0.0000
C01433=-96.515,22.174,78.476,-179.7076,-1.9027,0.0000
C01434=-95.839,28.477,78.891,179.9656,-0.1203,0.0000
C01435=-93.673,34.998,79.163,179.9943,-0.0115,0.0000
C01436=-90.984,41.489,79.163,179.9943,-0.0115,0.0000
C01437=-87.904,47.632,78.891,179.9370,-0.1089,0.0000
C01438=-83.926,52.567,78.476,178.4467,-1.1407,0.0000
C01439=-78.373,54.731,78.062,176.0662,-0.4480,0.0000
C01440=-72.396,53.692,77.551,174.3756,2.7184,0.0000
C01441=-66.782,49.709,76.575,174.8773,3.7188,0.0000
C01442=-60.870,45.159,74.567,175.5194,3.2487,0.0000
C01443=-55.523,41.042,71.901,176.4881,2.4691,0.0000
C01444=-51.344,38.042,69.285,178.8997,0.6992,0.0000
C01445=-48.211,36.955,67.386,-158.4444,1.3677,0.0000
C01446=-45.408,38.660,66.632,-152.8255,23.3683,0.0000
C01447=-43.572,40.607,66.599,-154.9221,26.9843,0.0000
C01448=-42.111,42.111,66.621,-153.9499,26.0501,0.0000
C01449=-40.607,43.571,66.599,-153.0102,25.0779,0.0000
C01450=-38.659,45.409,66.632,-156.6317,27.1745,0.0000
C01451=-36.955,48.211,67.386,-178.6384,21.5556,0.0000
C01452=-38.042,51.344,69.285,-179.3008,-1.1003,0.0000
C01453=-41.042,55.523,71.901,-177.5309,-3.5119,0.0000
C01454=-45.159,60.870,74.567,-176.7513,-4.4806,0.0000
C01455=-49.709,66.782,76.575,-176.2812,-5.1227,0.0000
C01456=-53.692,72.396,77.551,-177.2816,-5.6244,0.0000
C01457=-54.731,78.373,78.062,179.5520,-3.9338,0.0000
C01458=-52.567,83.926,78.476,178.8593,-1.5533,0.0000
C01459=-47.632,87.904,78.891,179.8911,-0.0630,0.0000
C01460=-41.489,90.984,79.163,179.9885,-0.0057,0.0000
C01461=-34.998,93.673,79.163,179.9885,-0.0057,0.0000
C01462=-28.477,95.839,78.891,179.8797,-0.0344,0.0000
C01463=-22.174,96.515,78.476,178.0973,0.2924,0.0000
C01464=-16.717,94.118,78.062,176.9016,2.4681,0.0000
C01465=-13.226,89.158,77.551,177.9318,5.8869,0.0000
C01466=-12.073,82.372,76.575,179.0028,6.2415,0.0000
C01467=-11.109,74.974,74.567,179.1251,5.4574,0.0000
C01468=-10.239,68.282,71.901,179.2646,4.2269,0.0000
C01469=-9.406,63.206,69.285,179.7192,1.2721,0.0000
C01470=-7.959,60.222,67.386,-163.5011,-14.7099,0.0000
C01471=-4.772,59.445,66.632,-146.2383,-3.2876,0.0000
C01472=-2.096,59.523,66.599,-145.3578,1.6714,0.0000
C01473=0.000,59.554,66.621,-145.3422,-0.0000,0.0000
C01474=0.000,58.319,68.442,-146.3576,-0.0000,0.0000
C01475=1.984,58.291,68.419,-146.3687,-1.5621,0.0000
C01476=4.582,58.225,68.453,-147.3220,3.5059,0.0000
C01477=7.730,59.058,69.238,-164.9129,14.0635,0.0000
C01478=9.135,62.185,71.215,179.6618,-1.6102,0.0000
C01479=9.949,67.473,73.927,179.3049,-4.1407,0.0000
C01480=10.820,74.409,76.674,179.2061,-5.1467,0.0000
C01481=11.787,82.032,78.729,179.1131,-5.7688,0.0000
C01482=12.929,88.996,79.725,178.1580,-5.4083,0.0000
C01483=16.445,94.085,80.245,177.1834,-2.2837,0.0000
C01484=21.964,96.553,80.665,178.2693,-0.2752,0.0000
C01485=28.347,95.882,81.086,179.8911,0.0344,0.0000
C01486=34.955,93.690,81.363,179.9885,0.0057,0.0000
C01487=41.532,90.965,81.363,179.9885,0.0057,0.0000
C01488=47.755,87.843,81.086,179.8969,0.0573,0.0000
C01489=52.743,83.804,80.665,178.9683,1.4156,0.0000
C01490=54.900,78.157,80.245,179.6211,3.6006,0.0000
C01491=53.787,72.072,79.725,-177.4680,5.1285,0.0000
C01492=49.670,66.340,78.729,-176.5427,4.7064,0.0000
C01493=44.964,60.266,76.674,-176.9193,4.2038,0.0000
C01494=40.676,54.746,73.927,-177.5598,3.4200,0.0000
C01495=37.512,50.430,71.215,-179.1002,1.3754,0.0000
C01496=36.294,47.226,69.238,-179.2247,-20.1946,0.0000
C01497=37.931,44.411,68.453,-157.6916,-26.4231,0.0000
C01498=39.816,42.621,68.419,-153.9105,-24.2804,0.0000
C01499=41.238,41.238,68.442,-154.7969,-25.2031,0.0000
C01500=42.621,39.816,68.419,-155.7196,-26.0895,0.0000
C01501=44.412,37.931,68.453,-153.5769,-22.3026,0.0000
C01502=47.226,36.294,69.238,-159.8054,-0.7753,0.0000
C01503=50.430,37.512,71.215,178.6246,-0.8998,0.0000
C01504=54.746,40.676,73.927,176.5800,-2.4402,0.0000
C01505=60.266,44.964,76.674,175.7962,-3.0807,0.0000
C01506=66.340,49.670,78.729,175.2936,-3.4573,0.0000
C01507=72.072,53.787,79.725,174.8715,-2.5320,0.0000
C01508=78.157,54.900,80.245,176.3994,0.3789,0.0000
C01509=83.804,52.743,80.665,178.5844,1.0317,0.0000
C01510=87.843,47.755,81.086,179.9427,0.1031,0.0000
C01511=90.965,41.532,81.363,179.9943,0.0115,0.0000
C01512=93.690,34.955,81.363,179.9943,0.0115,0.0000
C01513=95.882,28.347,81.086,179.9656,0.1089,0.0000
C01514=96.553,21.964,80.665,-179.7248,1.7307,0.0000
C01515=94.085,16.445,80.245,-177.7163,2.8166,0.0000
C01516=88.996,12.929,79.725,-174.5917,1.8420,0.0000
C01517=82.032,11.787,78.729,-174.2312,0.8869,0.0000
C01518=74.409,10.820,76.674,-174.8533,0.7939,0.0000
C01519=67.473,9.949,73.927,-175.8593,0.6951,0.0000
C01520=62.185,9.135,71.215,-178.3898,0.3382,0.0000
C01521=59.058,7.730,69.238,165.9365,-15.0871,0.0000
C01522=58.225,4.582,68.453,176.4941,-32.6780,0.0000
C01523=58.291,1.984,68.419,-178.4379,-33.6313,0.0000
C01524=58.319,0.000,68.442,-180.0000,-33.6424,0.0000
C01525=58.291,-1.983,68.419,178.4379,-33.6313,0.0000
C01526=58.225,-4.583,68.453,-176.4941,-32.6780,0.0000
C01527=59.058,-7.730,69.238,-165.9365,-15.0871,0.0000
C01528=62.185,-9.135,71.215,178.3898,0.3382,0.0000
C01529=67.473,-9.949,73.927,175.8593,0.6951,0.0000
C01530=74.409,-10.820,76.674,174.8533,0.7939,0.0000
C01531=82.032,-11.787,78.729,174.2312,0.8869,0.0000
C01532=88.996,-12.929,79.725,174.5917,1.8420,0.0000
C01533=94.085,-16.445,80.245,177.7163,2.8166,0.0000
C01534=96.553,-21.964,80.665,179.7248,1.7307,0.0000
C01535=95.882,-28.347,81.086,-179.9656,0.1089,0.0000
C01536=93.690,-34.955,81.363,-179.9943,0.0115,0.0000
C01537=90.965,-41.532,81.363,-179.9943,0.0115,0.0000
C01538=87.843,-47.755,81.086,-179.9427,0.1031,0.0000
C01539=83.804,-52.743,80.665,-178.5844,1.0317,0.0000
C01540=78.157,-54.900,80.245,-176.3994,0.3789,0.0000
C01541=72.072,-53.787,79.725,-174.8715,-2.5320,0.0000
C01542=66.340,-49.670,78.729,-175.2936,-3.4573,0.0000
C01543=60.266,-44.964,76.674,-175.7962,-3.0807,0.0000
C01544=54.746,-40.676,73.927,-176.5800,-2.4402,0.0000
C01545=50.430,-37.512,71.215,-178.6246,-0.8998,0.0000
C01546=47.226,-36.294,69.238,159.8054,-0.7753,0.0000
C01547=44.411,-37.931,68.453,153.5769,-22.3084,0.0000
C01548=42.621,-39.816,68.419,155.7196,-26.0895,0.0000
C01549=41.238,-41.238,68.442,154.7969,-25.2031,0.0000
C01550=39.816,-42.621,68.419,153.9105,-24.2804,0.0000
C01551=37.931,-44.412,68.453,157.6974,-26.4231,0.0000
C01552=36.294,-47.226,69.238,179.2247,-20.1946,0.0000
C01553=37.512,-50.430,71.215,179.1002,1.3754,0.0000
C01554=40.676,-54.746,73.927,177.5598,3.4200,0.0000
C01555=44.964,-60.266,76.674,176.9193,4.2038,0.0000
C01556=49.670,-66.340,78.729,176.5427,4.7064,0.0000
C01557=53.787,-72.072,79.725,177.4680,5.1285,0.0000
C01558=54.900,-78.157,80.245,-179.6211,3.6006,0.0000
C01559=52.743,-83.804,80.665,-178.9683,1.4156,0.0000
C01560=47.755,-87.843,81.086,-179.8969,0.0573,0.0000
C01561=41.532,-90.965,81.363,-179.9885,0.0057,0.0000
C01562=34.955,-93.690,81.363,-179.9885,0.0057,0.0000
C01563=28.347,-95.882,81.086,-179.8911,0.0344,0.0000
C01564=21.964,-96.553,80.665,-178.2693,-0.2752,0.0000
C01565=16.445,-94.085,80.245,-177.1834,-2.2837,0.0000
C01566=12.929,-88.996,79.725,-178.1580,-5.4083,0.0000
C01567=11.787,-82.032,78.729,-179.1131,-5.7688,0.0000
C01568=10.820,-74.409,76.674,-179.2061,-5.1467,0.0000
C01569=9.949,-67.473,73.927,-179.3049,-4.1407,0.0000
C01570=9.135,-62.185,71.215,-179.6618,-1.6102,0.0000
C01571=7.730,-59.058,69.238,164.9129,14.0635,0.0000
C01572=4.582,-58.225,68.453,147.3220,3.5059,0.0000
C01573=1.984,-58.291,68.419,146.3687,-1.5621,0.0000
C01574=0.000,-58.319,68.442,146.3576,-0.0000,0.0000
C01575=0.000,-58.319,68.442,146.3576,-0.0000,0.0000
C01576=-1.983,-58.291,68.419,146.3687,1.5621,0.0000
C01577=-4.583,-58.225,68.453,147.3220,-3.5059,0.0000
C01578=-7.730,-59.058,69.238,164.9129,-14.0635,0.0000
C01579=-9.135,-62.185,71.215,-179.6618,1.6102,0.0000
C01580=-9.949,-67.473,73.927,-179.3049,4.1407,0.0000
C01581=-10.820,-74.409,76.674,-179.2061,5.1467,0.0000
C01582=-11.787,-82.032,78.729,-179.1131,5.7688,0.0000
C01583=-12.929,-88.996,79.725,-178.1580,5.4083,0.0000
C01584=-16.445,-94.085,80.245,-177.1834,2.2837,0.0000
C01585=-21.964,-96.553,80.665,-178.2693,0.2752,0.0000
C01586=-28.347,-95.882,81.086,-179.8911,-0.0344,0.0000
C01587=-34.955,-93.690,81.363,-179.9885,-0.0057,0.0000
C01588=-41.532,-90.965,81.363,-179.9885,-0.0057,0.0000
C01589=-47.755,-87.843,81.086,-179.8969,-0.0573,0.0000
C01590=-52.743,-83.804,80.665,-178.9683,-1.4156,0.0000
C01591=-54.900,-78.157,80.245,-179.6211,-3.6006,0.0000
C01592=-53.787,-72.072,79.725,177.4680,-5.1285,0.0000
C01593=-49.670,-66.340,78.729,176.5427,-4.7064,0.0000
C01594=-44.964,-60.266,76.674,176.9193,-4.2038,0.0000
C01595=-40.676,-54.746,73.927,177.5598,-3.4200,0.0000
C01596=-37.512,-50.430,71.215,179.1002,-1.3754,0.0000
C01597=-36.294,-47.226,69.238,179.2247,20.1946,0.0000
C01598=-37.931,-44.411,68.453,157.6916,26.4231,0.0000
C01599=-39.816,-42.621,68.419,153.9105,24.2804,0.0000
C01600=-41.238,-41.238,68.442,154.7969,25.2031,0.0000
C01601=-42.621,-39.816,68.419,155.7196,26.0895,0.0000
C01602=-44.412,-37.931,68.453,153.5769,22.3026,0.0000
C01603=-47.226,-36.294,69.238,159.8054,0.7753,0.0000
C01604=-50.430,-37.512,71.215,-178.6246,0.8998,0.0000
C01605=-54.746,-40.676,73.927,-176.5800,2.4402,0.0000
C01606=-60.266,-44.964,76.674,-175.7962,3.0807,0.0000
C01607=-66.340,-49.670,78.729,-175.2936,3.4573,0.0000
C01608=-72.072,-53.787,79.725,-174.8715,2.5320,0.0000
C01609=-78.157,-54.900,80.245,-176.3994,-0.3789,0.0000
C01610=-83.804,-52.743,80.665,-178.5844,-1.0317,0.0000
C01611=-87.843,-47.755,81.086,-179.9427,-0.1031,0.0000
C01612=-90.965,-41.532,81.363,-179.9943,-0.0115,0.0000
C01613=-93.690,-34.955,81.363,-179.9943,-0.0115,0.0000
C01614=-95.882,-28.347,81.086,-179.9656,-0.1089,0.0000
C01615=-96.553,-21.964,80.665,179.7248,-1.7307,0.0000
C01616=-94.085,-16.445,80.245,177.7163,-2.8166,0.0000
C01617=-88.996,-12.929,79.725,174.5917,-1.8420,0.0000
C01618=-82.032,-11.787,78.729,174.2312,-0.8869,0.0000
C01619=-74.409,-10.820,76.674,174.8533,-0.7939,0.0000
C01620=-67.473,-9.949,73.927,175.8593,-0.6951,0.0000
C01621=-62.185,-9.135,71.215,178.3898,-0.3382,0.0000
C01622=-59.058,-7.730,69.238,-165.9365,15.0871,0.0000
C01623=-58.225,-4.582,68.453,-176.4941,32.6780,0.0000
C01624=-58.291,-1.984,68.419,178.4379,33.6313,0.0000
C01625=-58.319,0.000,68.442,180.0000,33.6424,0.0000
C01626=-58.291,1.983,68.419,-178.4379,33.6313,0.0000
C01627=-58.225,4.583,68.453,176.4941,32.6780,0.0000
C01628=-59.058,7.730,69.238,165.9365,15.0871,0.0000
C01629=-62.185,9.135,71.215,-178.3898,-0.3382,0.0000
C01630=-67.473,9.949,73.927,-175.8593,-0.6951,0.0000
C01631=-74.409,10.820,76.674,-174.8533,-0.7939,0.0000
C01632=-82.032,11.787,78.729,-174.2312,-0.8869,0.0000
C01633=-88.996,12.929,79.725,-174.5917,-1.8420,0.0000
C01634=-94.085,16.445,80.245,-177.7163,-2.8166,0.0000
C01635=-96.553,21.964,80.665,-179.7248,-1.7307,0.0000
C01636=-95.882,28.347,81.086,179.9656,-0.1089,0.0000
C01637=-93.690,34.955,81.363,179.9943,-0.0115,0.0000
C01638=-90.965,41.532,81.363,179.9943,-0.0115,0.0000
C01639=-87.843,47.755,81.086,179.9427,-0.1031,0.0000
C01640=-83.804,52.743,80.665,178.5844,-1.0317,0.0000
C01641=-78.157,54.900,80.245,176.3994,-0.3789,0.0000
C01642=-72.072,53.787,79.725,174.8715,2.5320,0.0000
C01643=-66.340,49.670,78.729,175.2936,3.4573,0.0000
C01644=-60.266,44.964,76.674,175.7962,3.0807,0.0000
C01645=-54.746,40.676,73.927,176.5800,2.4402,0.0000
C01646=-50.430,37.512,71.215,178.6246,0.8998,0.0000
C01647=-47.226,36.294,69.238,-159.8054,0.7753,0.0000
C01648=-44.411,37.931,68.453,-153.5769,22.3084,0.0000
C01649=-42.621,39.816,68.419,-155.7196,26.0895,0.0000
C01650=-41.238,41.238,68.442,-154.7969,25.2031,0.0000
C01651=-39.816,42.621,68.419,-153.9105,24.2804,0.0000
C01652=-37.931,44.412,68.453,-157.6974,26.4231,0.0000
C01653=-36.294,47.226,69.238,-179.2247,20.1946,0.0000
C01654=-37.512,50.430,71.215,-179.1002,-1.3754,0.0000
C01655=-40.676,54.746,73.927,-177.5598,-3.4200,0.0000
C01656=-44.964,60.266,76.674,-176.9193,-4.2038,0.0000
C01657=-49.670,66.340,78.729,-176.5427,-4.7064,0.0000
C01658=-53.787,72.072,79.725,-177.4680,-5.1285,0.0000
C01659=-54.900,78.157,80.245,179.6211,-3.6006,0.0000
C01660=-52.743,83.804,80.665,178.9683,-1.4156,0.0000
C01661=-47.755,87.843,81.086,179.8969,-0.0573,0.0000
C01662=-41.532,90.965,81.363,179.9885,-0.0057,0.0000
C01663=-34.955,93.690,81.363,179.9885,-0.0057,0.0000
C01664=-28.347,95.882,81.086,179.8911,-0.0344,0.0000
C01665=-21.964,96.553,80.665,178.2693,0.2752,0.0000
C01666=-16.445,94.085,80.245,177.1834,2.2837,0.0000
C01667=-12.929,88.996,79.725,178.1580,5.4083,0.0000
C01668=-11.787,82.032,78.729,179.1131,5.7688,0.0000
C01669=-10.820,74.409,76.674,179.2061,5.1467,0.0000
C01670=-9.949,67.473,73.927,179.3049,4.1407,0.0000
C01671=-9.135,62.185,71.215,179.6618,1.6102,0.0000
C01672=-7.730,59.058,69.238,-164.9129,-14.0635,0.0000
C01673=-4.583,58.225,68.453,-147.3220,-3.5059,0.0000
C01674=-1.983,58.291,68.419,-146.3687,1.5621,0.0000
C01675=0.000,58.319,68.442,-146.3576,-0.0000,0.0000
C01676=0.000,57.118,70.285,-147.5051,-0.0000,0.0000
C01677=1.874,57.094,70.261,-147.5117,-1.4401,0.0000
C01678=4.398,57.039,70.297,-148.5402,3.6814,0.0000
C01679=7.507,57.930,71.114,-166.2875,13.3407,0.0000
C01680=8.875,61.204,73.167,179.6331,-1.8624,0.0000
C01681=9.674,66.709,75.971,179.3567,-3.9970,0.0000
C01682=10.553,73.885,78.794,179.2871,-4.7727,0.0000
C01683=11.527,81.722,80.892,179.2232,-5.2333,0.0000
C01684=12.662,88.851,81.904,178.3840,-4.8665,0.0000
C01685=16.202,94.056,82.431,177.4938,-2.0593,0.0000
C01686=21.776,96.587,82.857,178.4585,-0.2522,0.0000
C01687=28.231,95.920,83.283,179.9026,0.0286,0.0000
C01688=34.916,93.705,83.562,179.9885,0.0057,0.0000
C01689=41.570,90.949,83.562,179.9885,0.0057,0.0000
C01690=47.863,87.788,83.283,179.9083,0.0516,0.0000
C01691=52.900,83.695,82.857,179.0887,1.2665,0.0000
C01692=55.051,77.964,82.431,179.6844,3.2275,0.0000
C01693=53.873,71.781,81.904,-177.6945,4.5865,0.0000
C01694=49.635,65.937,80.892,-176.8441,4.2504,0.0000
C01695=44.783,59.707,78.794,-177.1218,3.8866,0.0000
C01696=40.330,54.011,75.971,-177.6234,3.2819,0.0000
C01697=37.003,49.553,73.167,-178.9396,1.5760,0.0000
C01698=35.654,46.271,71.114,-179.7216,-18.7901,0.0000
C01699=37.223,43.442,70.297,-158.8323,-25.5526,0.0000
C01700=39.047,41.697,70.261,-154.9184,-23.3869,0.0000
C01701=40.388,40.388,70.285,-155.7514,-24.2486,0.0000
C01702=41.696,39.047,70.261,-156.6131,-25.0816,0.0000
C01703=43.443,37.223,70.297,-154.4474,-21.1618,0.0000
C01704=46.271,35.654,71.114,-161.2099,-0.2784,0.0000
C01705=49.553,37.003,73.167,178.4240,-1.0604,0.0000
C01706=54.011,40.330,75.971,176.7181,-2.3766,0.0000
C01707=59.707,44.783,78.794,176.1134,-2.8782,0.0000
C01708=65.937,49.635,80.892,175.7496,-3.1559,0.0000
C01709=71.781,53.873,81.904,175.4135,-2.3055,0.0000
C01710=77.964,55.051,82.431,176.7725,0.3156,0.0000
C01711=83.695,52.900,82.857,178.7335,0.9113,0.0000
C01712=87.788,47.863,83.283,179.9484,0.0917,0.0000
C01713=90.949,41.570,83.562,179.9943,0.0115,0.0000
C01714=93.705,34.916,83.562,179.9943,0.0115,0.0000
C01715=95.920,28.231,83.283,179.9714,0.0974,0.0000
C01716=96.587,21.776,82.857,-179.7478,1.5415,0.0000
C01717=94.056,16.202,82.431,-177.9407,2.5062,0.0000
C01718=88.851,12.662,81.904,-175.1335,1.6160,0.0000
C01719=81.722,11.527,80.892,-174.7667,0.7768,0.0000
C01720=73.885,10.553,78.794,-175.2273,0.7129,0.0000
C01721=66.709,9.674,75.971,-176.0030,0.6433,0.0000
C01722=61.204,8.875,73.167,-178.1376,0.3669,0.0000
C01723=57.930,7.507,71.114,166.6593,-13.7125,0.0000
C01724=57.039,4.398,70.297,176.3186,-31.4598,0.0000
C01725=57.094,1.874,70.261,-178.5599,-32.4883,0.0000
C01726=57.118,0.000,70.285,-180.0000,-32.4949,0.0000
C01727=57.094,-1.874,70.261,178.5599,-32.4883,0.0000
C01728=57.039,-4.398,70.297,-176.3186,-31.4598,0.0000
C01729=57.930,-7.507,71.114,-166.6593,-13.7125,0.0000
C01730=61.204,-8.875,73.167,178.1376,0.3669,0.0000
C01731=66.709,-9.674,75.971,176.0030,0.6433,0.0000
C01732=73.885,-10.553,78.794,175.2273,0.7129,0.0000
C01733=81.722,-11.527,80.892,174.7667,0.7768,0.0000
C01734=88.851,-12.662,81.904,175.1335,1.6160,0.0000
C01735=94.056,-16.202,82.431,177.9407,2.5062,0.0000
C01736=96.587,-21.776,82.857,179.7478,1.5415,0.0000
C01737=95.920,-28.231,83.283,-179.9714,0.0974,0.0000
C01738=93.705,-34.916,83.562,-179.9943,0.0115,0.0000
C01739=90.949,-41.570,83.562,-179.9943,0.0115,0.0000
C01740=87.788,-47.863,83.283,-179.9484,0.0917,0.0000
C01741=83.695,-52.900,82.857,-178.7335,0.9113,0.0000
C01742=77.964,-55.051,82.431,-176.7725,0.3156,0.0000
C01743=71.781,-53.873,81.904,-175.4135,-2.3055,0.0000
C01744=65.937,-49.635,80.892,-175.7496,-3.1559,0.0000
C01745=59.707,-44.783,78.794,-176.1134,-2.8782,0.0000
C01746=54.011,-40.330,75.971,-176.7181,-2.3766,0.0000
C01747=49.553,-37.003,73.167,-178.4240,-1.0604,0.0000
C01748=46.271,-35.654,71.114,161.2099,-0.2784,0.0000
C01749=43.442,-37.223,70.297,154.4474,-21.1677,0.0000
C01750=41.697,-39.047,70.261,156.6131,-25.0816,0.0000
C01751=40.388,-40.388,70.285,155.7514,-24.2486,0.0000
C01752=39.047,-41.696,70.261,154.9184,-23.3869,0.0000
C01753=37.223,-43.443,70.297,158.8382,-25.5526,0.0000
C01754=35.654,-46.271,71.114,179.7216,-18.7901,0.0000
C01755=37.003,-49.553,73.167,178.9396,1.5760,0.0000
C01756=40.330,-54.011,75.971,177.6234,3.2819,0.0000
C01757=44.783,-59.707,78.794,177.1218,3.8866,0.0000
C01758=49.635,-65.937,80.892,176.8441,4.2504,0.0000
C01759=53.873,-71.781,81.904,177.6945,4.5865,0.0000
C01760=55.051,-77.964,82.431,-179.6844,3.2275,0.0000
C01761=52.900,-83.695,82.857,-179.0887,1.2665,0.0000
C01762=47.863,-87.788,83.283,-179.9083,0.0516,0.0000
C01763=41.570,-90.949,83.562,-179.9885,0.0057,0.0000
C01764=34.916,-93.705,83.562,-179.9885,0.0057,0.0000
C01765=28.231,-95.920,83.283,-179.9026,0.0286,0.0000
C01766=21.776,-96.587,82.857,-178.4585,-0.2522,0.0000
C01767=16.202,-94.056,82.431,-177.4938,-2.0593,0.0000
C01768=12.662,-88.851,81.904,-178.3840,-4.8665,0.0000
C01769=11.527,-81.722,80.892,-179.2232,-5.2333,0.0000
C01770=10.553,-73.885,78.794,-179.2871,-4.7727,0.0000
C01771=9.674,-66.709,75.971,-179.3567,-3.9970,0.0000
C01772=8.875,-61.204,73.167,-179.6331,-1.8624,0.0000
C01773=7.507,-57.930,71.114,166.2875,13.3407,0.0000
C01774=4.398,-57.039,70.297,148.5402,3.6814,0.0000
C01775=1.874,-57.094,70.261,147.5117,-1.4401,0.0000
C01776=0.000,-57.118,70.285,147.5051,-0.0000,0.0000
C01777=0.000,-57.118,70.285,147.5051,-0.0000,0.0000
C01778=-1.874,-57.094,70.261,147.5117,1.4401,0.0000
C01779=-4.398,-57.039,70.297,148.5402,-3.6814,0.0000
C01780=-7.507,-57.930,71.114,166.2875,-13.3407,0.0000
C01781=-8.875,-61.204,73.167,-179.6331,1.8624,0.0000
C01782=-9.674,-66.709,75.971,-179.3567,3.9970,0.0000
C01783=-10.553,-73.885,78.794,-179.2871,4.7727,0.0000
C01784=-11.527,-81.722,80.892,-179.2232,5.2333,0.0000
C01785=-12.662,-88.851,81.904,-178.3840,4.8665,0.0000
C01786=-16.202,-94.056,82.431,-177.4938,2.0593,0.0000
C01787=-21.776,-96.587,82.857,-178.4585,0.2522,0.0000
C01788=-28.231,-95.920,83.283,-179.9026,-0.0286,0.0000
C01789=-34.916,-93.705,83.562,-179.9885,-0.0057,0.0000
C01790=-41.570,-90.949,83.562,-179.9885,-0.0057,0.0000
C01791=-47.863,-87.788,83.283,-179.9083,-0.0516,0.0000
C01792=-52.900,-83.695,82.857,-179.0887,-1.2665,0.0000
C01793=-55.051,-77.964,82.431,-179.6844,-3.2275,0.0000
C01794=-53.873,-71.781,81.904,177.6945,-4.5865,0.0000
C01795=-49.635,-65.937,80.892,176.8441,-4.2504,0.0000
C01796=-44.783,-59.707,78.794,177.1218,-3.8866,0.0000
C01797=-40.330,-54.011,75.971,177.6234,-3.2819,0.0000
C01798=-37.003,-49.553,73.167,178.9396,-1.5760,0.0000
C01799=-35.654,-46.271,71.114,179.7216,18.7901,0.0000
C01800=-37.223,-43.442,70.297,158.8323,25.5526,0.0000
C01801=-39.047,-41.697,70.261,154.9184,23.3869,0.0000
C01802=-40.388,-40.388,70.285,155.7514,24.2486,0.0000
C01803=-41.696,-39.047,70.261,156.6131,25.0816,0.0000
C01804=-43.443,-37.223,70.297,154.4474,21.1618,0.0000
C01805=-46.271,-35.654,71.114,161.2099,0.2784,0.0000
C01806=-49.553,-37.003,73.167,-178.4240,1.0604,0.0000
C01807=-54.011,-40.330,75.971,-176.7181,2.3766,0.0000
C01808=-59.707,-44.783,78.794,-176.1134,2.8782,0.0000
C01809=-65.937,-49.635,80.892,-175.7496,3.1559,0.0000
C01810=-71.781,-53.873,81.904,-175.4135,2.3055,0.0000
C01811=-77.964,-55.051,82.431,-176.7725,-0.3156,0.0000
C01812=-83.695,-52.900,82.857,-178.7335,-0.9113,0.0000
C01813=-87.788,-47.863,83.283,-179.9484,-0.0917,0.0000
C01814=-90.949,-41.570,83.562,-179.9943,-0.0115,0.0000
C01815=-93.705,-34.916,83.562,-179.9943,-0.0115,0.0000
C01816=-95.920,-28.231,83.283,-179.9714,-0.0974,0.0000
C01817=-96.587,-21.776,82.857,179.7478,-1.5415,0.0000
C01818=-94.056,-16.202,82.431,177.9407,-2.5062,0.0000
C01819=-88.851,-12.662,81.904,175.1335,-1.6160,0.0000
C01820=-81.722,-11.527,80.892,174.7667,-0.7768,0.0000
C01821=-73.885,-10.553,78.794,175.2273,-0.7129,0.0000
C01822=-66.709,-9.674,75.971,176.0030,-0.6433,0.0000
C01823=-61.204,-8.875,73.167,178.1376,-0.3669,0.0000
C01824=-57.930,-7.507,71.114,-166.6593,13.7125,0.0000
C01825=-57.039,-4.398,70.297,-176.3186,31.4598,0.0000
C01826=-57.094,-1.874,70.261,178.5599,32.4883,0.0000
C01827=-57.118,0.000,70.285,180.0000,32.4949,0.0000
C01828=-57.094,1.874,70.261,-178.5599,32.4883,0.0000
C01829=-57.039,4.398,70.297,176.3186,31.4598,0.0000
C01830=-57.930,7.507,71.114,166.6593,13.7125,0.0000
C01831=-61.204,8.875,73.167,-178.1376,-0.3669,0.0000
C01832=-66.709,9.674,75.971,-176.0030,-0.6433,0.0000
C01833=-73.885,10.553,78.794,-175.2273,-0.7129,0.0000
C01834=-81.722,11.527,80.892,-174.7667,-0.7768,0.0000
C01835=-88.851,12.662,81.904,-175.1335,-1.6160,0.0000
C01836=-94.056,16.202,82.431,-177.9407,-2.5062,0.0000
C01837=-96.587,21.776,82.857,-179.7478,-1.5415,0.0000
C01838=-95.920,28.231,83.283,179.9714,-0.0974,0.0000
C01839=-93.705,34.916,83.562,179.9943,-0.0115,0.0000
C01840=-90.949,41.570,83.562,179.9943,-0.0115,0.0000
C01841=-87.788,47.863,83.283,179.9484,-0.0917,0.0000
C01842=-83.695,52.900,82.857,178.7335,-0.9113,0.0000
C01843=-77.964,55.051,82.431,176.7725,-0.3156,0.0000
C01844=-71.781,53.873,81.904,175.4135,2.3055,0.0000
C01845=-65.937,49.635,80.892,175.7496,3.1559,0.0000
C01846=-59.707,44.783,78.794,176.1134,2.8782,0.0000
C01847=-54.011,40.330,75.971,176.7181,2.3766,0.0000
C01848=-49.553,37.003,73.167,178.4240,1.0604,0.0000
C01849=-46.271,35.654,71.114,-161.2099,0.2784,0.0000
C01850=-43.442,37.223,70.297,-154.4474,21.1677,0.0000
C01851=-41.697,39.047,70.261,-156.6131,25.0816,0.0000
C01852=-40.388,40.388,70.285,-155.7514,24.2486,0.0000
C01853=-39.047,41.696,70.261,-154.9184,23.3869,0.0000
C01854=-37.223,43.443,70.297,-158.8382,25.5526,0.0000
C01855=-35.654,46.271,71.114,-179.7216,18.7901,0.0000
C01856=-37.003,49.553,73.167,-178.9396,-1.5760,0.0000
C01857=-40.330,54.011,75.971,-177.6234,-3.2819,0.0000
C01858=-44.783,59.707,78.794,-177.1218,-3.8866,0.0000
C01859=-49.635,65.937,80.892,-176.8441,-4.2504,0.0000
C01860=-53.873,71.781,81.904,-177.6945,-4.5865,0.0000
C01861=-55.051,77.964,82.431,179.6844,-3.2275,0.0000
C01862=-52.900,83.695,82.857,179.0887,-1.2665,0.0000
C01863=-47.863,87.788,83.283,179.9083,-0.0516,0.0000
C01864=-41.570,90.949,83.562,179.9885,-0.0057,0.0000
C01865=-34.916,93.705,83.562,179.9885,-0.0057,0.0000
C01866=-28.231,95.920,83.283,179.9026,-0.0286,0.0000
C01867=-21.776,96.587,82.857,178.4585,0.2522,0.0000
C01868=-16.202,94.056,82.431,177.4938,2.0593,0.0000
C01869=-12.662,88.851,81.904,178.3840,4.8665,0.0000
C01870=-11.527,81.722,80.892,179.2232,5.2333,0.0000
C01871=-10.553,73.885,78.794,179.2871,4.7727,0.0000
C01872=-9.674,66.709,75.971,179.3567,3.9970,0.0000
C01873=-8.875,61.204,73.167,179.6331,1.8624,0.0000
C01874=-7.507,57.930,71.114,-166.2875,-13.3407,0.0000
C01875=-4.398,57.039,70.297,-148.5402,-3.6814,0.0000
C01876=-1.874,57.094,70.261,-147.5117,1.4401,0.0000
C01877=0.000,57.118,70.285,-147.5051,-0.0000,0.0000
